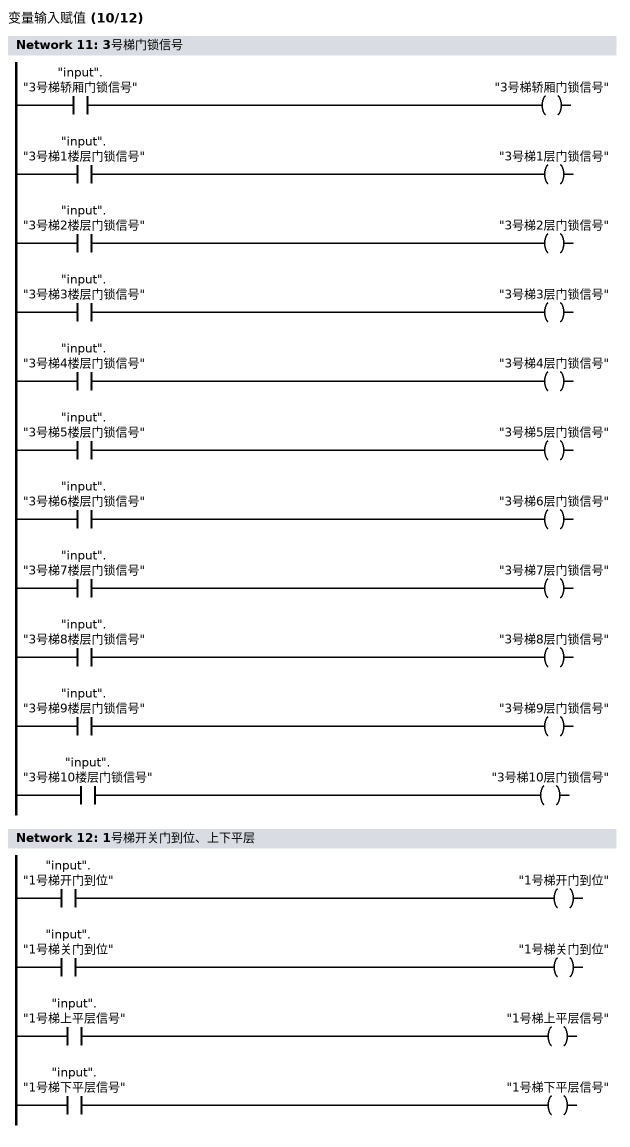
   RUNG wire#powerrail
      Contact( "input"."3号梯轿厢门锁信号" )
      Coil( "3号梯轿厢门锁信号" )
   END_RUNG
   RUNG wire#powerrail
      Contact( "input"."3号梯1楼层门锁信号" )
      Coil( "3号梯1层门锁信号" )
   END_RUNG
   RUNG wire#powerrail
      Contact( "input"."3号梯2楼层门锁信号" )
      Coil( "3号梯2层门锁信号" )
   END_RUNG
   RUNG wire#powerrail
      Contact( "input"."3号梯3楼层门锁信号" )
      Coil( "3号梯3层门锁信号" )
   END_RUNG
   RUNG wire#powerrail
      Contact( "input"."3号梯4楼层门锁信号" )
      Coil( "3号梯4层门锁信号" )
   END_RUNG
   RUNG wire#powerrail
      Contact( "input"."3号梯5楼层门锁信号" )
      Coil( "3号梯5层门锁信号" )
   END_RUNG
   RUNG wire#powerrail
      Contact( "input"."3号梯6楼层门锁信号" )
      Coil( "3号梯6层门锁信号" )
   END_RUNG
   RUNG wire#powerrail
      Contact( "input"."3号梯7楼层门锁信号" )
      Coil( "3号梯7层门锁信号" )
   END_RUNG
   RUNG wire#powerrail
      Contact( "input"."3号梯8楼层门锁信号" )
      Coil( "3号梯8层门锁信号" )
   END_RUNG
   RUNG wire#powerrail
      Contact( "input"."3号梯9楼层门锁信号" )
      Coil( "3号梯9层门锁信号" )
   END_RUNG
   RUNG wire#powerrail
      Contact( "input"."3号梯10楼层门锁信号" )
      Coil( "3号梯10层门锁信号" )
   END_RUNG
   // the same network as SCL:
   "3号梯轿厢门锁信号" := "input"."3号梯轿厢门锁信号";
   "3号梯1层门锁信号" := "input"."3号梯1楼层门锁信号";
   "3号梯2层门锁信号" := "input"."3号梯2楼层门锁信号";
   "3号梯3层门锁信号" := "input"."3号梯3楼层门锁信号";
   "3号梯4层门锁信号" := "input"."3号梯4楼层门锁信号";
   "3号梯5层门锁信号" := "input"."3号梯5楼层门锁信号";
   "3号梯6层门锁信号" := "input"."3号梯6楼层门锁信号";
   "3号梯7层门锁信号" := "input"."3号梯7楼层门锁信号";
   "3号梯8层门锁信号" := "input"."3号梯8楼层门锁信号";
   "3号梯9层门锁信号" := "input"."3号梯9楼层门锁信号";
   "3号梯10层门锁信号" := "input"."3号梯10楼层门锁信号";
END_REGION

REGION Network 12: 1号梯开关门到位、上下平层
   RUNG wire#powerrail
      Contact( "input"."1号梯开门到位" )
      Coil( "1号梯开门到位" )
   END_RUNG
   RUNG wire#powerrail
      Contact( "input"."1号梯关门到位" )
      Coil( "1号梯关门到位" )
   END_RUNG
   RUNG wire#powerrail
      Contact( "input"."1号梯上平层信号" )
      Coil( "1号梯上平层信号" )
   END_RUNG
   RUNG wire#powerrail
      Contact( "input"."1号梯下平层信号" )
      Coil( "1号梯下平层信号" )
   END_RUNG
   // the same network as SCL:
   "1号梯开门到位" := "input"."1号梯开门到位";
   "1号梯关门到位" := "input"."1号梯关门到位";
   "1号梯上平层信号" := "input"."1号梯上平层信号";
   "1号梯下平层信号" := "input"."1号梯下平层信号";
END_REGION

REGION Network 13: 2号梯开关门到位、上下平层
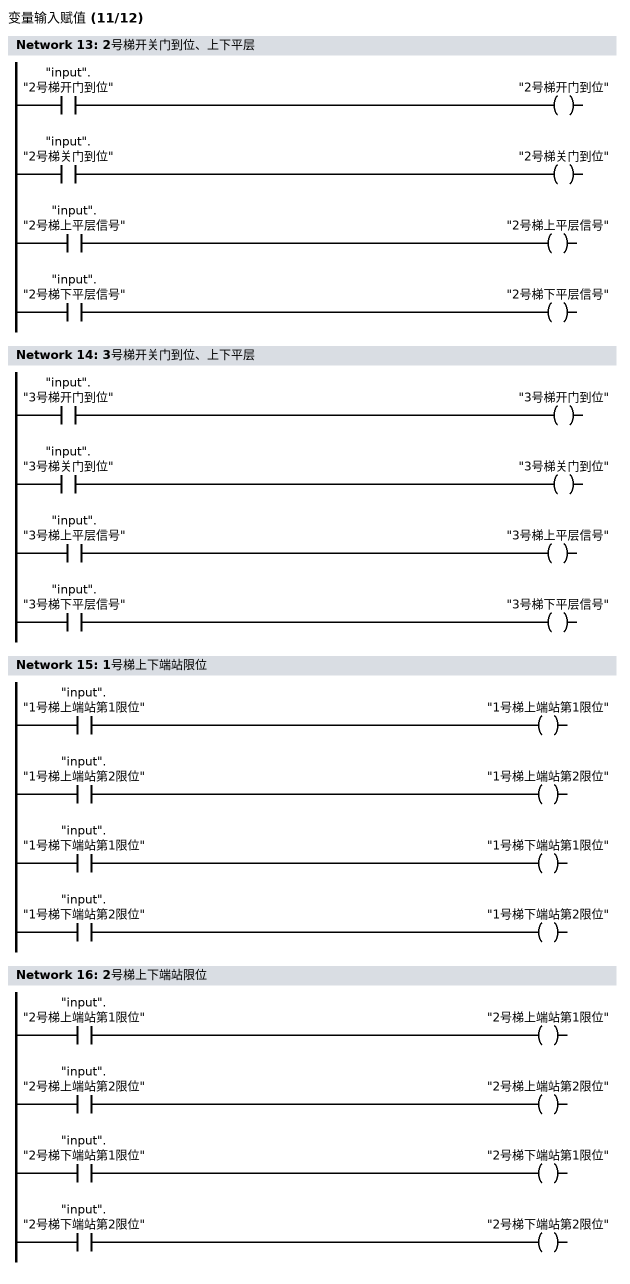
   RUNG wire#powerrail
      Contact( "input"."2号梯开门到位" )
      Coil( "2号梯开门到位" )
   END_RUNG
   RUNG wire#powerrail
      Contact( "input"."2号梯关门到位" )
      Coil( "2号梯关门到位" )
   END_RUNG
   RUNG wire#powerrail
      Contact( "input"."2号梯上平层信号" )
      Coil( "2号梯上平层信号" )
   END_RUNG
   RUNG wire#powerrail
      Contact( "input"."2号梯下平层信号" )
      Coil( "2号梯下平层信号" )
   END_RUNG
   // the same network as SCL:
   "2号梯开门到位" := "input"."2号梯开门到位";
   "2号梯关门到位" := "input"."2号梯关门到位";
   "2号梯上平层信号" := "input"."2号梯上平层信号";
   "2号梯下平层信号" := "input"."2号梯下平层信号";
END_REGION

REGION Network 14: 3号梯开关门到位、上下平层
   RUNG wire#powerrail
      Contact( "input"."3号梯开门到位" )
      Coil( "3号梯开门到位" )
   END_RUNG
   RUNG wire#powerrail
      Contact( "input"."3号梯关门到位" )
      Coil( "3号梯关门到位" )
   END_RUNG
   RUNG wire#powerrail
      Contact( "input"."3号梯上平层信号" )
      Coil( "3号梯上平层信号" )
   END_RUNG
   RUNG wire#powerrail
      Contact( "input"."3号梯下平层信号" )
      Coil( "3号梯下平层信号" )
   END_RUNG
   // the same network as SCL:
   "3号梯开门到位" := "input"."3号梯开门到位";
   "3号梯关门到位" := "input"."3号梯关门到位";
   "3号梯上平层信号" := "input"."3号梯上平层信号";
   "3号梯下平层信号" := "input"."3号梯下平层信号";
END_REGION

REGION Network 15: 1号梯上下端站限位
   RUNG wire#powerrail
      Contact( "input"."1号梯上端站第1限位" )
      Coil( "1号梯上端站第1限位" )
   END_RUNG
   RUNG wire#powerrail
      Contact( "input"."1号梯上端站第2限位" )
      Coil( "1号梯上端站第2限位" )
   END_RUNG
   RUNG wire#powerrail
      Contact( "input"."1号梯下端站第1限位" )
      Coil( "1号梯下端站第1限位" )
   END_RUNG
   RUNG wire#powerrail
      Contact( "input"."1号梯下端站第2限位" )
      Coil( "1号梯下端站第2限位" )
   END_RUNG
   // the same network as SCL:
   "1号梯上端站第1限位" := "input"."1号梯上端站第1限位";
   "1号梯上端站第2限位" := "input"."1号梯上端站第2限位";
   "1号梯下端站第1限位" := "input"."1号梯下端站第1限位";
   "1号梯下端站第2限位" := "input"."1号梯下端站第2限位";
END_REGION

REGION Network 16: 2号梯上下端站限位
   RUNG wire#powerrail
      Contact( "input"."2号梯上端站第1限位" )
      Coil( "2号梯上端站第1限位" )
   END_RUNG
   RUNG wire#powerrail
      Contact( "input"."2号梯上端站第2限位" )
      Coil( "2号梯上端站第2限位" )
   END_RUNG
   RUNG wire#powerrail
      Contact( "input"."2号梯下端站第1限位" )
      Coil( "2号梯下端站第1限位" )
   END_RUNG
   RUNG wire#powerrail
      Contact( "input"."2号梯下端站第2限位" )
      Coil( "2号梯下端站第2限位" )
   END_RUNG
   // the same network as SCL:
   "2号梯上端站第1限位" := "input"."2号梯上端站第1限位";
   "2号梯上端站第2限位" := "input"."2号梯上端站第2限位";
   "2号梯下端站第1限位" := "input"."2号梯下端站第1限位";
   "2号梯下端站第2限位" := "input"."2号梯下端站第2限位";
END_REGION

REGION Network 17: 3号梯上下端站限位
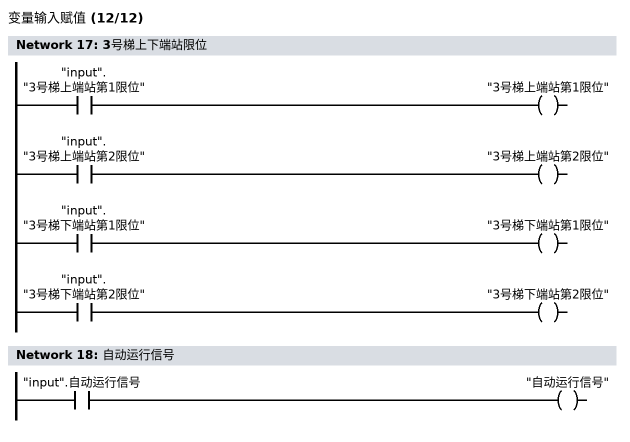
   RUNG wire#powerrail
      Contact( "input"."3号梯上端站第1限位" )
      Coil( "3号梯上端站第1限位" )
   END_RUNG
   RUNG wire#powerrail
      Contact( "input"."3号梯上端站第2限位" )
      Coil( "3号梯上端站第2限位" )
   END_RUNG
   RUNG wire#powerrail
      Contact( "input"."3号梯下端站第1限位" )
      Coil( "3号梯下端站第1限位" )
   END_RUNG
   RUNG wire#powerrail
      Contact( "input"."3号梯下端站第2限位" )
      Coil( "3号梯下端站第2限位" )
   END_RUNG
   // the same network as SCL:
   "3号梯上端站第1限位" := "input"."3号梯上端站第1限位";
   "3号梯上端站第2限位" := "input"."3号梯上端站第2限位";
   "3号梯下端站第1限位" := "input"."3号梯下端站第1限位";
   "3号梯下端站第2限位" := "input"."3号梯下端站第2限位";
END_REGION

REGION Network 18: 自动运行信号
   RUNG wire#powerrail
      Contact( "input".自动运行信号 )
      Coil( "自动运行信号" )
   END_RUNG
   // the same network as SCL:
   "自动运行信号" := "input".自动运行信号;
END_REGION
END_FUNCTION

FUNCTION "FC_GC_Score" : Int   // FC4, SCL
{ S7_Optimized_Access := 'TRUE' }
   VAR_INPUT
      ReqFloor : Int;
      ReqDir : Int;
      LiftFloor : Int;
      LiftDir : Int;
      LiftRunning : Bool;
      LiftLoadPercent : Int;
      TaskCount : Int;
      AheadTaskCount : Int;
      CanUse : Bool;
      W_Distance : Int;
      W_Direction : Int;
      W_Task : Int;
      W_AheadTask : Int;
      W_LoadPercent : Real;
      empty : Int;
   END_VAR
   VAR_TEMP
      tmpDist : Int;
      tmpScore : Int;
   END_VAR
BEGIN
   // ==================================================
   // FC_GC_Score 优化版
   //
   // 方向定义：
   //    1 = 上行
   //    0 = 停止/空闲
   //   -1 = 下行
   //
   // 评分越低，派梯优先级越高
   // ==================================================


   // ==================================================
   // 1. 可用性及输入有效性检查
   // ==================================================
   IF (NOT #CanUse)
       OR (#ReqFloor < 1)
       OR (#ReqFloor > 10)
       OR (#LiftFloor < 1)
       OR (#LiftFloor > 10)
       OR ((#ReqDir <> 1) AND (#ReqDir <> -1))
       OR (
       (#LiftDir <> -1)
       AND (#LiftDir <> 0)
       AND (#LiftDir <> 1)
       ) THEN

       // 32000表示该电梯不可参与派梯
       #FC_GC_Score := 32000;

   ELSE

       // ==================================================
       // 2. 距离评分
       // ==================================================
       #tmpDist := ABS(#ReqFloor - #LiftFloor);

       #tmpScore :=
       #tmpDist * #W_Distance;


       // ==================================================
       // 3. 方向和路线评分
       // ==================================================

       // --------------------------------------------------
       // 3.1 LiftDir = 0：停止或空闲
       // --------------------------------------------------
       IF #LiftDir = 0 THEN

           // 所有方向为0的电梯均获得空闲奖励
           // 不限制电梯所在楼层
           #tmpScore :=
           #tmpScore - #empty;


           // --------------------------------------------------
           // 3.2 电梯运行方向与外呼方向相同
           // --------------------------------------------------
       ELSIF #LiftDir = #ReqDir THEN

           // 上行梯：请求楼层在当前楼层上方或同层
           // 下行梯：请求楼层在当前楼层下方或同层
           IF
               (
               (#LiftDir = 1)
               AND (#ReqFloor >= #LiftFloor)
               )
               OR
               (
               (#LiftDir = -1)
               AND (#ReqFloor <= #LiftFloor)
               ) THEN

               // 同方向且请求在运行前方，属于顺路
               #tmpScore := #tmpScore + 0;

           ELSE

               // 方向相同，但是已经越过请求楼层
               // 必须完成当前路线后换向返回
               #tmpScore :=
               #tmpScore
               + (#W_Direction * 2);

               // 增加部分返回距离惩罚
               #tmpScore :=
               #tmpScore
               + (
               #tmpDist
               * #W_Distance
               / 2
               );

           END_IF;


           // --------------------------------------------------
           // 3.3 电梯运行方向与外呼方向相反
           // --------------------------------------------------
       ELSE

           // 判断请求楼层是否位于电梯当前运动前方
           IF
               (
               (#LiftDir = 1)
               AND (#ReqFloor >= #LiftFloor)
               )
               OR
               (
               (#LiftDir = -1)
               AND (#ReqFloor <= #LiftFloor)
               ) THEN

               // 请求楼层位于当前运行前方，
               // 但是乘客请求方向与电梯方向相反
               #tmpScore :=
               #tmpScore
               + (#W_Direction * 2);

           ELSE

               // 请求楼层位于当前运行后方，
               // 同时乘客请求方向也与电梯方向相反
               // 属于最不利的派梯情况
               #tmpScore :=
               #tmpScore
               + (#W_Direction * 3);

               // 增加部分绕行距离惩罚
               #tmpScore :=
               #tmpScore
               + (
               #tmpDist
               * #W_Distance
               / 2
               );

           END_IF;

       END_IF;


       // ==================================================
       // 4. 当前总任务数量惩罚
       // ==================================================
       IF #TaskCount > 0 THEN

           #tmpScore :=
           #tmpScore
           + (#TaskCount * #W_Task);

       END_IF;


       // ==================================================
       // 5. 当前运行前方任务数量惩罚
       // ==================================================
       IF #AheadTaskCount > 0 THEN

           #tmpScore :=
           #tmpScore
           + (
           #AheadTaskCount
           * #W_AheadTask
           );

       END_IF;


       // ==================================================
       // 6. 载重量基础评分
       // ==================================================
       IF #LiftLoadPercent > 0 THEN

           #tmpScore :=
           #tmpScore
           + REAL_TO_INT(
                         INT_TO_REAL(#LiftLoadPercent)
                         * #W_LoadPercent
           );

       END_IF;


       // ==================================================
       // 7. 高载重附加惩罚
       // ==================================================
       IF #LiftLoadPercent >= 90 THEN

           // 载重量达到90%以上
           #tmpScore :=
           #tmpScore + #W_Direction;

       ELSIF #LiftLoadPercent >= 75 THEN

           // 载重量达到75%以上
           #tmpScore :=
           #tmpScore + (#W_Direction / 2);

       END_IF;


       // ==================================================
       // 8. 同层空闲电梯额外奖励
       // ==================================================
       IF (#tmpDist = 0)
           AND (#LiftDir = 0) THEN

           // 已经获得普通空闲奖励，
           // 同层空闲时再增加一次奖励
           #tmpScore :=
           #tmpScore
           - (#W_Direction / 2);

       END_IF;


       // ==================================================
       // 9. 最终评分范围保护
       // ==================================================
       IF #tmpScore < 0 THEN

           #tmpScore := 0;

       ELSIF #tmpScore > 31999 THEN

           // 32000专门保留给不可用电梯
           #tmpScore := 31999;

       END_IF;


       // ==================================================
       // 10. 返回评分结果
       // ==================================================
       #FC_GC_Score := #tmpScore;

   END_IF;
END_FUNCTION

FUNCTION "FC_GC_IO_Map" : Void   // FC5, SCL
{ S7_Optimized_Access := 'TRUE' }
BEGIN
      // ==================================================
      // 1. 鏃犳晥妤煎眰淇濇姢
      // ==================================================
      "DB_GC".HallUpBtn[10] := FALSE;
      "DB_GC".HallDownBtn[1] := FALSE;


      // ==================================================
      // 2. 鏆傛椂娌℃湁杞藉鐜囧拰鍔熺巼锛屽氨鍏堢粰榛樿鍊?
       // ==================================================
      "DB_GC".LiftLoadPercent[1] := 0;
      "DB_GC".LiftLoadPercent[2] := 0;
      "DB_GC".LiftLoadPercent[3] := 0;

      "DB_GC".LiftPower_kW[1] := 0.0;
      "DB_GC".LiftPower_kW[2] := 0.0;
      "DB_GC".LiftPower_kW[3] := 0.0;


      // ==================================================
      // 3. 缇ゆ帶浣胯兘 / 閿佹 / 绂佺敤
      // 鍚庨潰鎺?WINCC 鏃跺啀鏀规垚 HMI 鍙橀噺
      // ==================================================
      "DB_GC".LiftGroupEnable[1] := TRUE;
      "DB_GC".LiftGroupEnable[2] := TRUE;
      "DB_GC".LiftGroupEnable[3] := TRUE;

      "DB_GC".LiftLocked[1] := FALSE;
      "DB_GC".LiftLocked[2] := FALSE;
      "DB_GC".LiftLocked[3] := FALSE;

      "DB_GC".LiftDisabled[1] := FALSE;
      "DB_GC".LiftDisabled[2] := FALSE;
      "DB_GC".LiftDisabled[3] := FALSE;


      // ==================================================
      // 4. 缇ゆ帶妯″紡
      // 0鏅€氾紝1涓婄彮楂樺嘲锛?涓嬬彮楂樺嘲锛?鍗堥楂樺嘲锛?涓夊垎鍖?
       // ==================================================
      "DB_GC".GroupMode := 0;


      // ==================================================
      // 5. 涔樻鏃堕棿缁熻锛屾殏鏃朵笉鐢?
       // ==================================================
      "DB_GC".RideFinishPulse[1] := FALSE;
      "DB_GC".RideFinishPulse[2] := FALSE;
      "DB_GC".RideFinishPulse[3] := FALSE;

      "DB_GC".RideTimeSample_s[1] := 0.0;
      "DB_GC".RideTimeSample_s[2] := 0.0;
      "DB_GC".RideTimeSample_s[3] := 0.0;
END_FUNCTION

FUNCTION "消防模式" : Void   // FC6, LAD
{ S7_Optimized_Access := 'TRUE' }
VERSION : 0.1
   VAR_TEMP   // added for the SCL form of the ladder/FBD networks
      _w1 : Bool;
   END_VAR
BEGIN

REGION Network 1: 指示灯reset
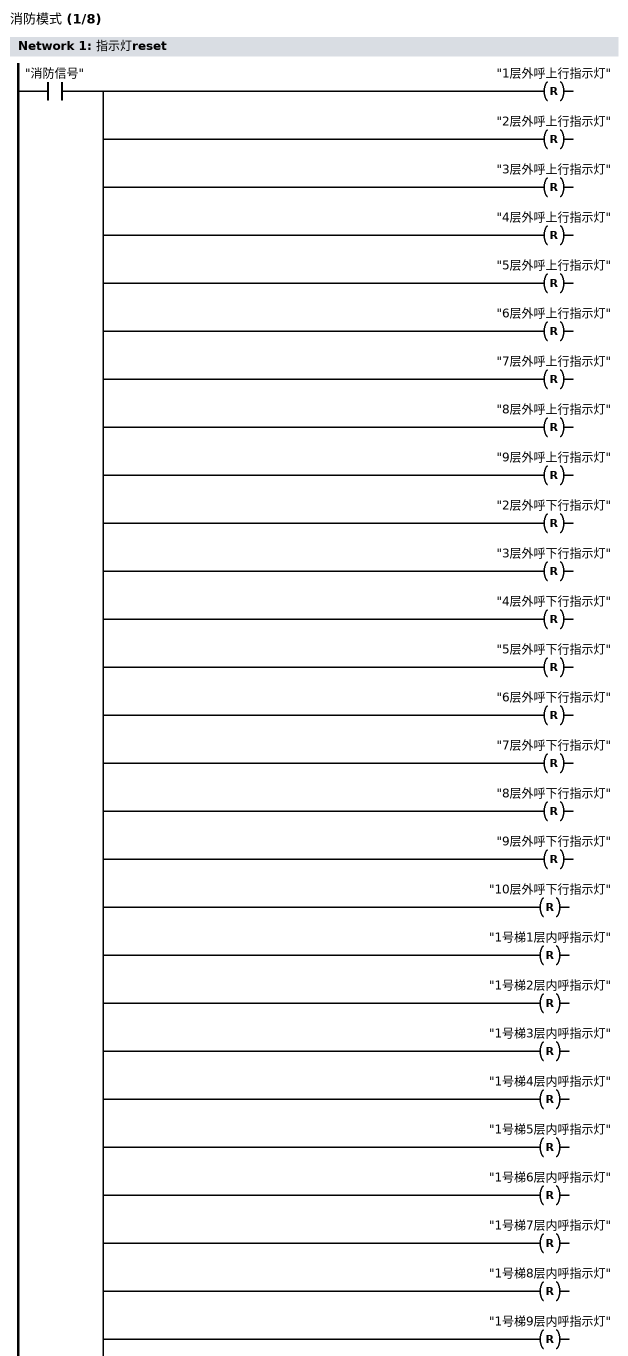
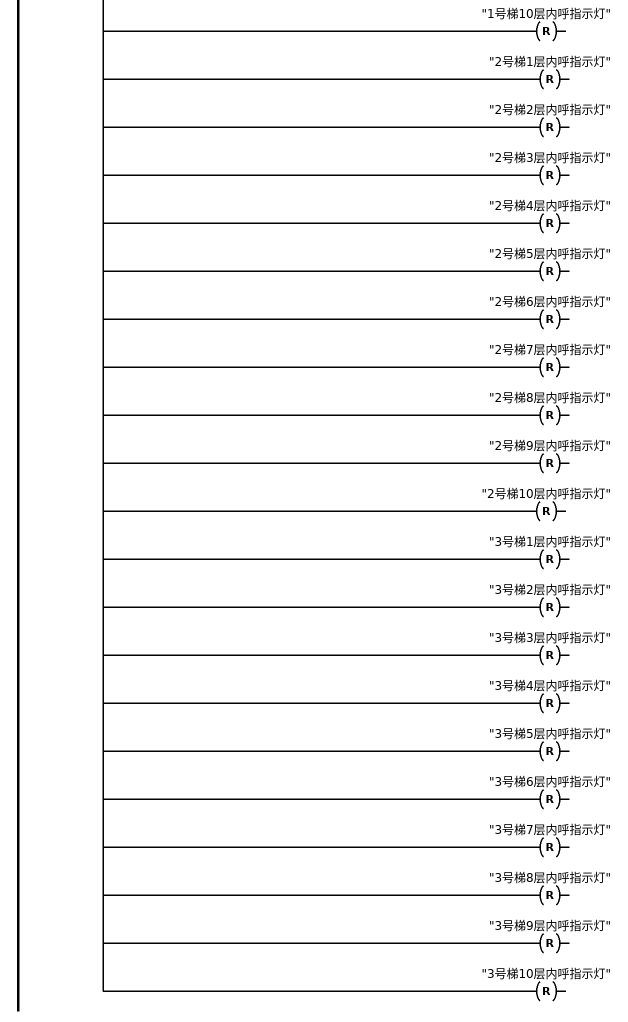
   RUNG wire#powerrail
      Contact( "消防信号" )
      wire#w1
      R_Coil( "1层外呼上行指示灯" )
   END_RUNG
   RUNG wire#w1
      R_Coil( "2层外呼上行指示灯" )
   END_RUNG
   RUNG wire#w1
      R_Coil( "3层外呼上行指示灯" )
   END_RUNG
   RUNG wire#w1
      R_Coil( "4层外呼上行指示灯" )
   END_RUNG
   RUNG wire#w1
      R_Coil( "5层外呼上行指示灯" )
   END_RUNG
   RUNG wire#w1
      R_Coil( "6层外呼上行指示灯" )
   END_RUNG
   RUNG wire#w1
      R_Coil( "7层外呼上行指示灯" )
   END_RUNG
   RUNG wire#w1
      R_Coil( "8层外呼上行指示灯" )
   END_RUNG
   RUNG wire#w1
      R_Coil( "9层外呼上行指示灯" )
   END_RUNG
   RUNG wire#w1
      R_Coil( "2层外呼下行指示灯" )
   END_RUNG
   RUNG wire#w1
      R_Coil( "3层外呼下行指示灯" )
   END_RUNG
   RUNG wire#w1
      R_Coil( "4层外呼下行指示灯" )
   END_RUNG
   RUNG wire#w1
      R_Coil( "5层外呼下行指示灯" )
   END_RUNG
   RUNG wire#w1
      R_Coil( "6层外呼下行指示灯" )
   END_RUNG
   RUNG wire#w1
      R_Coil( "7层外呼下行指示灯" )
   END_RUNG
   RUNG wire#w1
      R_Coil( "8层外呼下行指示灯" )
   END_RUNG
   RUNG wire#w1
      R_Coil( "9层外呼下行指示灯" )
   END_RUNG
   RUNG wire#w1
      R_Coil( "10层外呼下行指示灯" )
   END_RUNG
   RUNG wire#w1
      R_Coil( "1号梯1层内呼指示灯" )
   END_RUNG
   RUNG wire#w1
      R_Coil( "1号梯2层内呼指示灯" )
   END_RUNG
   RUNG wire#w1
      R_Coil( "1号梯3层内呼指示灯" )
   END_RUNG
   RUNG wire#w1
      R_Coil( "1号梯4层内呼指示灯" )
   END_RUNG
   RUNG wire#w1
      R_Coil( "1号梯5层内呼指示灯" )
   END_RUNG
   RUNG wire#w1
      R_Coil( "1号梯6层内呼指示灯" )
   END_RUNG
   RUNG wire#w1
      R_Coil( "1号梯7层内呼指示灯" )
   END_RUNG
   RUNG wire#w1
      R_Coil( "1号梯8层内呼指示灯" )
   END_RUNG
   RUNG wire#w1
      R_Coil( "1号梯9层内呼指示灯" )
   END_RUNG
   RUNG wire#w1
      R_Coil( "1号梯10层内呼指示灯" )
   END_RUNG
   RUNG wire#w1
      R_Coil( "2号梯1层内呼指示灯" )
   END_RUNG
   RUNG wire#w1
      R_Coil( "2号梯2层内呼指示灯" )
   END_RUNG
   RUNG wire#w1
      R_Coil( "2号梯3层内呼指示灯" )
   END_RUNG
   RUNG wire#w1
      R_Coil( "2号梯4层内呼指示灯" )
   END_RUNG
   RUNG wire#w1
      R_Coil( "2号梯5层内呼指示灯" )
   END_RUNG
   RUNG wire#w1
      R_Coil( "2号梯6层内呼指示灯" )
   END_RUNG
   RUNG wire#w1
      R_Coil( "2号梯7层内呼指示灯" )
   END_RUNG
   RUNG wire#w1
      R_Coil( "2号梯8层内呼指示灯" )
   END_RUNG
   RUNG wire#w1
      R_Coil( "2号梯9层内呼指示灯" )
   END_RUNG
   RUNG wire#w1
      R_Coil( "2号梯10层内呼指示灯" )
   END_RUNG
   RUNG wire#w1
      R_Coil( "3号梯1层内呼指示灯" )
   END_RUNG
   RUNG wire#w1
      R_Coil( "3号梯2层内呼指示灯" )
   END_RUNG
   RUNG wire#w1
      R_Coil( "3号梯3层内呼指示灯" )
   END_RUNG
   RUNG wire#w1
      R_Coil( "3号梯4层内呼指示灯" )
   END_RUNG
   RUNG wire#w1
      R_Coil( "3号梯5层内呼指示灯" )
   END_RUNG
   RUNG wire#w1
      R_Coil( "3号梯6层内呼指示灯" )
   END_RUNG
   RUNG wire#w1
      R_Coil( "3号梯7层内呼指示灯" )
   END_RUNG
   RUNG wire#w1
      R_Coil( "3号梯8层内呼指示灯" )
   END_RUNG
   RUNG wire#w1
      R_Coil( "3号梯9层内呼指示灯" )
   END_RUNG
   RUNG wire#w1
      R_Coil( "3号梯10层内呼指示灯" )
   END_RUNG
   // the same network as SCL:
   IF "消防信号" THEN
       "1层外呼上行指示灯" := FALSE;
       "2层外呼上行指示灯" := FALSE;
       "3层外呼上行指示灯" := FALSE;
       "4层外呼上行指示灯" := FALSE;
       "5层外呼上行指示灯" := FALSE;
       "6层外呼上行指示灯" := FALSE;
       "7层外呼上行指示灯" := FALSE;
       "8层外呼上行指示灯" := FALSE;
       "9层外呼上行指示灯" := FALSE;
       "2层外呼下行指示灯" := FALSE;
       "3层外呼下行指示灯" := FALSE;
       "4层外呼下行指示灯" := FALSE;
       "5层外呼下行指示灯" := FALSE;
       "6层外呼下行指示灯" := FALSE;
       "7层外呼下行指示灯" := FALSE;
       "8层外呼下行指示灯" := FALSE;
       "9层外呼下行指示灯" := FALSE;
       "10层外呼下行指示灯" := FALSE;
       "1号梯1层内呼指示灯" := FALSE;
       "1号梯2层内呼指示灯" := FALSE;
       "1号梯3层内呼指示灯" := FALSE;
       "1号梯4层内呼指示灯" := FALSE;
       "1号梯5层内呼指示灯" := FALSE;
       "1号梯6层内呼指示灯" := FALSE;
       "1号梯7层内呼指示灯" := FALSE;
       "1号梯8层内呼指示灯" := FALSE;
       "1号梯9层内呼指示灯" := FALSE;
       "1号梯10层内呼指示灯" := FALSE;
       "2号梯1层内呼指示灯" := FALSE;
       "2号梯2层内呼指示灯" := FALSE;
       "2号梯3层内呼指示灯" := FALSE;
       "2号梯4层内呼指示灯" := FALSE;
       "2号梯5层内呼指示灯" := FALSE;
       "2号梯6层内呼指示灯" := FALSE;
       "2号梯7层内呼指示灯" := FALSE;
       "2号梯8层内呼指示灯" := FALSE;
       "2号梯9层内呼指示灯" := FALSE;
       "2号梯10层内呼指示灯" := FALSE;
       "3号梯1层内呼指示灯" := FALSE;
       "3号梯2层内呼指示灯" := FALSE;
       "3号梯3层内呼指示灯" := FALSE;
       "3号梯4层内呼指示灯" := FALSE;
       "3号梯5层内呼指示灯" := FALSE;
       "3号梯6层内呼指示灯" := FALSE;
       "3号梯7层内呼指示灯" := FALSE;
       "3号梯8层内呼指示灯" := FALSE;
       "3号梯9层内呼指示灯" := FALSE;
       "3号梯10层内呼指示灯" := FALSE;
   END_IF;
END_REGION

REGION Network 2: 群控输出reset
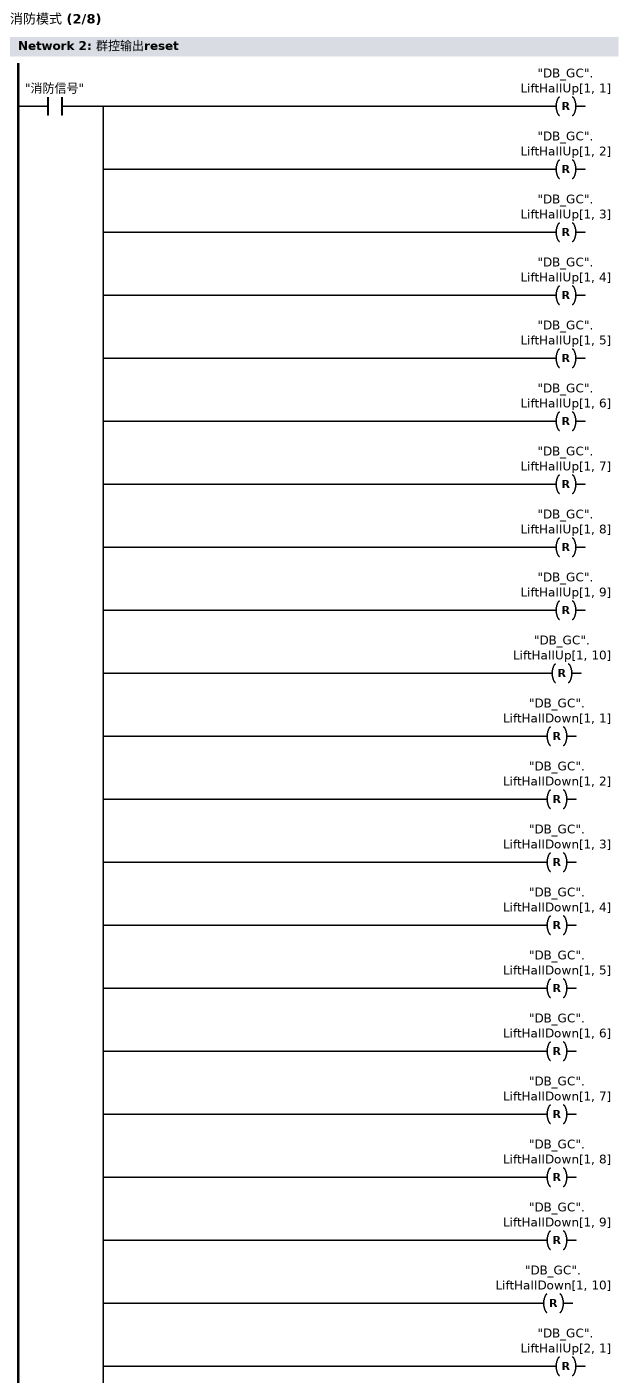
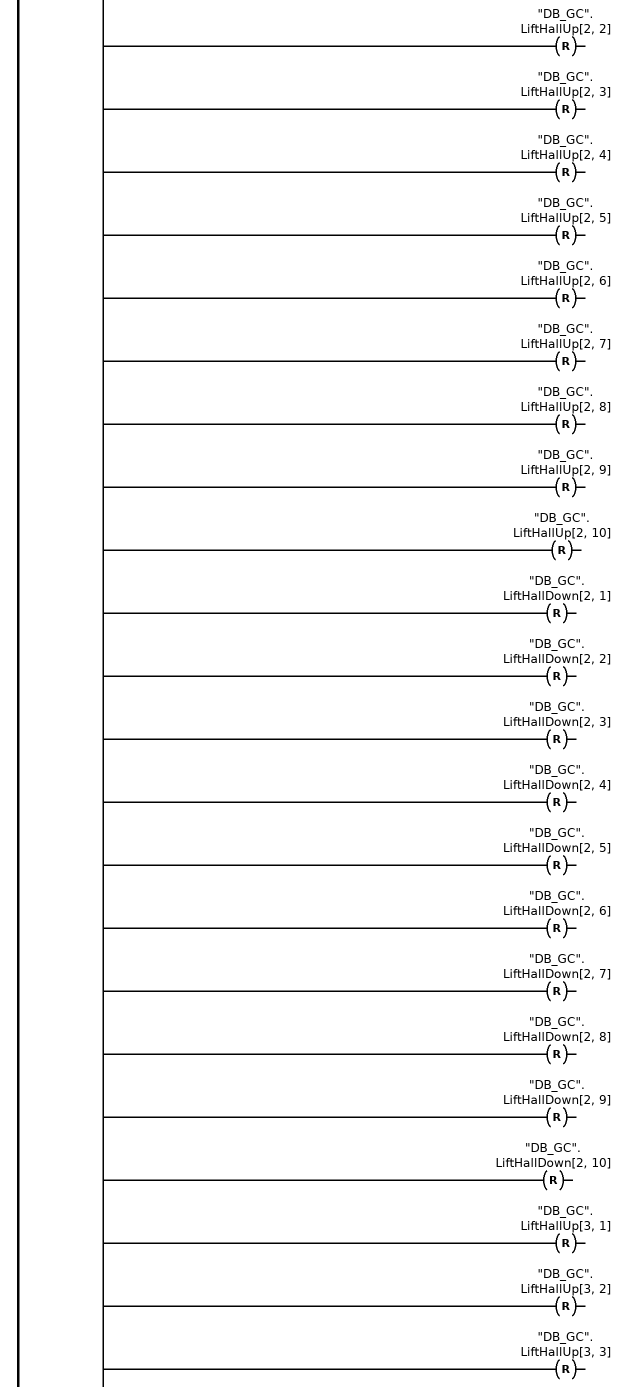
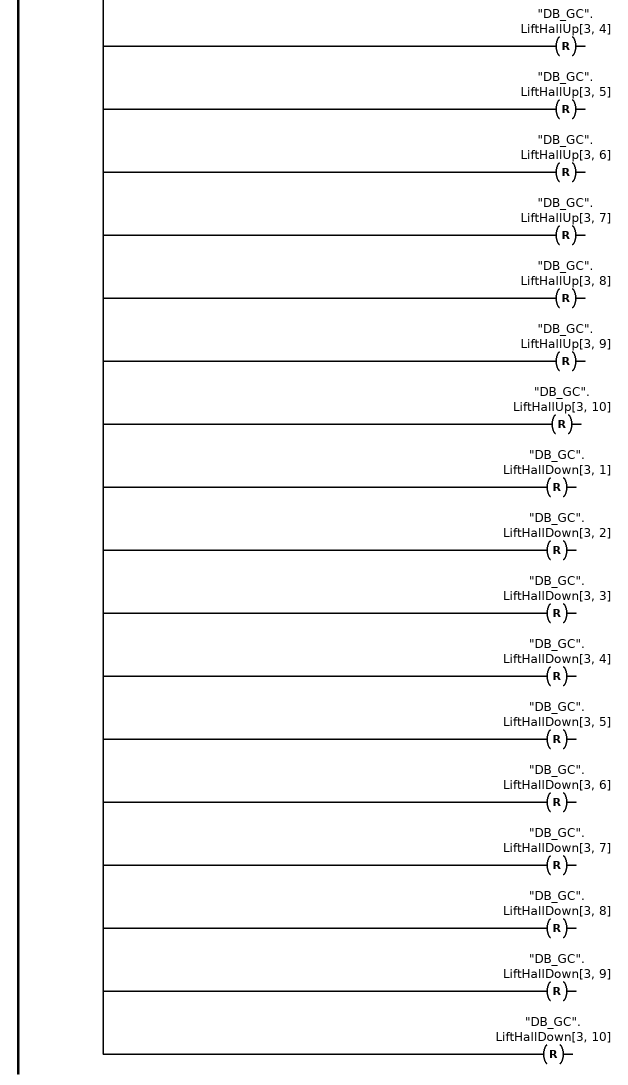
   RUNG wire#powerrail
      Contact( "消防信号" )
      wire#w1
      R_Coil( "DB_GC".LiftHallUp[1, 1] )
   END_RUNG
   RUNG wire#w1
      R_Coil( "DB_GC".LiftHallUp[1, 2] )
   END_RUNG
   RUNG wire#w1
      R_Coil( "DB_GC".LiftHallUp[1, 3] )
   END_RUNG
   RUNG wire#w1
      R_Coil( "DB_GC".LiftHallUp[1, 4] )
   END_RUNG
   RUNG wire#w1
      R_Coil( "DB_GC".LiftHallUp[1, 5] )
   END_RUNG
   RUNG wire#w1
      R_Coil( "DB_GC".LiftHallUp[1, 6] )
   END_RUNG
   RUNG wire#w1
      R_Coil( "DB_GC".LiftHallUp[1, 7] )
   END_RUNG
   RUNG wire#w1
      R_Coil( "DB_GC".LiftHallUp[1, 8] )
   END_RUNG
   RUNG wire#w1
      R_Coil( "DB_GC".LiftHallUp[1, 9] )
   END_RUNG
   RUNG wire#w1
      R_Coil( "DB_GC".LiftHallUp[1, 10] )
   END_RUNG
   RUNG wire#w1
      R_Coil( "DB_GC".LiftHallDown[1, 1] )
   END_RUNG
   RUNG wire#w1
      R_Coil( "DB_GC".LiftHallDown[1, 2] )
   END_RUNG
   RUNG wire#w1
      R_Coil( "DB_GC".LiftHallDown[1, 3] )
   END_RUNG
   RUNG wire#w1
      R_Coil( "DB_GC".LiftHallDown[1, 4] )
   END_RUNG
   RUNG wire#w1
      R_Coil( "DB_GC".LiftHallDown[1, 5] )
   END_RUNG
   RUNG wire#w1
      R_Coil( "DB_GC".LiftHallDown[1, 6] )
   END_RUNG
   RUNG wire#w1
      R_Coil( "DB_GC".LiftHallDown[1, 7] )
   END_RUNG
   RUNG wire#w1
      R_Coil( "DB_GC".LiftHallDown[1, 8] )
   END_RUNG
   RUNG wire#w1
      R_Coil( "DB_GC".LiftHallDown[1, 9] )
   END_RUNG
   RUNG wire#w1
      R_Coil( "DB_GC".LiftHallDown[1, 10] )
   END_RUNG
   RUNG wire#w1
      R_Coil( "DB_GC".LiftHallUp[2, 1] )
   END_RUNG
   RUNG wire#w1
      R_Coil( "DB_GC".LiftHallUp[2, 2] )
   END_RUNG
   RUNG wire#w1
      R_Coil( "DB_GC".LiftHallUp[2, 3] )
   END_RUNG
   RUNG wire#w1
      R_Coil( "DB_GC".LiftHallUp[2, 4] )
   END_RUNG
   RUNG wire#w1
      R_Coil( "DB_GC".LiftHallUp[2, 5] )
   END_RUNG
   RUNG wire#w1
      R_Coil( "DB_GC".LiftHallUp[2, 6] )
   END_RUNG
   RUNG wire#w1
      R_Coil( "DB_GC".LiftHallUp[2, 7] )
   END_RUNG
   RUNG wire#w1
      R_Coil( "DB_GC".LiftHallUp[2, 8] )
   END_RUNG
   RUNG wire#w1
      R_Coil( "DB_GC".LiftHallUp[2, 9] )
   END_RUNG
   RUNG wire#w1
      R_Coil( "DB_GC".LiftHallUp[2, 10] )
   END_RUNG
   RUNG wire#w1
      R_Coil( "DB_GC".LiftHallDown[2, 1] )
   END_RUNG
   RUNG wire#w1
      R_Coil( "DB_GC".LiftHallDown[2, 2] )
   END_RUNG
   RUNG wire#w1
      R_Coil( "DB_GC".LiftHallDown[2, 3] )
   END_RUNG
   RUNG wire#w1
      R_Coil( "DB_GC".LiftHallDown[2, 4] )
   END_RUNG
   RUNG wire#w1
      R_Coil( "DB_GC".LiftHallDown[2, 5] )
   END_RUNG
   RUNG wire#w1
      R_Coil( "DB_GC".LiftHallDown[2, 6] )
   END_RUNG
   RUNG wire#w1
      R_Coil( "DB_GC".LiftHallDown[2, 7] )
   END_RUNG
   RUNG wire#w1
      R_Coil( "DB_GC".LiftHallDown[2, 8] )
   END_RUNG
   RUNG wire#w1
      R_Coil( "DB_GC".LiftHallDown[2, 9] )
   END_RUNG
   RUNG wire#w1
      R_Coil( "DB_GC".LiftHallDown[2, 10] )
   END_RUNG
   RUNG wire#w1
      R_Coil( "DB_GC".LiftHallUp[3, 1] )
   END_RUNG
   RUNG wire#w1
      R_Coil( "DB_GC".LiftHallUp[3, 2] )
   END_RUNG
   RUNG wire#w1
      R_Coil( "DB_GC".LiftHallUp[3, 3] )
   END_RUNG
   RUNG wire#w1
      R_Coil( "DB_GC".LiftHallUp[3, 4] )
   END_RUNG
   RUNG wire#w1
      R_Coil( "DB_GC".LiftHallUp[3, 5] )
   END_RUNG
   RUNG wire#w1
      R_Coil( "DB_GC".LiftHallUp[3, 6] )
   END_RUNG
   RUNG wire#w1
      R_Coil( "DB_GC".LiftHallUp[3, 7] )
   END_RUNG
   RUNG wire#w1
      R_Coil( "DB_GC".LiftHallUp[3, 8] )
   END_RUNG
   RUNG wire#w1
      R_Coil( "DB_GC".LiftHallUp[3, 9] )
   END_RUNG
   RUNG wire#w1
      R_Coil( "DB_GC".LiftHallUp[3, 10] )
   END_RUNG
   RUNG wire#w1
      R_Coil( "DB_GC".LiftHallDown[3, 1] )
   END_RUNG
   RUNG wire#w1
      R_Coil( "DB_GC".LiftHallDown[3, 2] )
   END_RUNG
   RUNG wire#w1
      R_Coil( "DB_GC".LiftHallDown[3, 3] )
   END_RUNG
   RUNG wire#w1
      R_Coil( "DB_GC".LiftHallDown[3, 4] )
   END_RUNG
   RUNG wire#w1
      R_Coil( "DB_GC".LiftHallDown[3, 5] )
   END_RUNG
   RUNG wire#w1
      R_Coil( "DB_GC".LiftHallDown[3, 6] )
   END_RUNG
   RUNG wire#w1
      R_Coil( "DB_GC".LiftHallDown[3, 7] )
   END_RUNG
   RUNG wire#w1
      R_Coil( "DB_GC".LiftHallDown[3, 8] )
   END_RUNG
   RUNG wire#w1
      R_Coil( "DB_GC".LiftHallDown[3, 9] )
   END_RUNG
   RUNG wire#w1
      R_Coil( "DB_GC".LiftHallDown[3, 10] )
   END_RUNG
   // the same network as SCL:
   IF "消防信号" THEN
       "DB_GC".LiftHallUp[1, 1] := FALSE;
       "DB_GC".LiftHallUp[1, 2] := FALSE;
       "DB_GC".LiftHallUp[1, 3] := FALSE;
       "DB_GC".LiftHallUp[1, 4] := FALSE;
       "DB_GC".LiftHallUp[1, 5] := FALSE;
       "DB_GC".LiftHallUp[1, 6] := FALSE;
       "DB_GC".LiftHallUp[1, 7] := FALSE;
       "DB_GC".LiftHallUp[1, 8] := FALSE;
       "DB_GC".LiftHallUp[1, 9] := FALSE;
       "DB_GC".LiftHallUp[1, 10] := FALSE;
       "DB_GC".LiftHallDown[1, 1] := FALSE;
       "DB_GC".LiftHallDown[1, 2] := FALSE;
       "DB_GC".LiftHallDown[1, 3] := FALSE;
       "DB_GC".LiftHallDown[1, 4] := FALSE;
       "DB_GC".LiftHallDown[1, 5] := FALSE;
       "DB_GC".LiftHallDown[1, 6] := FALSE;
       "DB_GC".LiftHallDown[1, 7] := FALSE;
       "DB_GC".LiftHallDown[1, 8] := FALSE;
       "DB_GC".LiftHallDown[1, 9] := FALSE;
       "DB_GC".LiftHallDown[1, 10] := FALSE;
       "DB_GC".LiftHallUp[2, 1] := FALSE;
       "DB_GC".LiftHallUp[2, 2] := FALSE;
       "DB_GC".LiftHallUp[2, 3] := FALSE;
       "DB_GC".LiftHallUp[2, 4] := FALSE;
       "DB_GC".LiftHallUp[2, 5] := FALSE;
       "DB_GC".LiftHallUp[2, 6] := FALSE;
       "DB_GC".LiftHallUp[2, 7] := FALSE;
       "DB_GC".LiftHallUp[2, 8] := FALSE;
       "DB_GC".LiftHallUp[2, 9] := FALSE;
       "DB_GC".LiftHallUp[2, 10] := FALSE;
       "DB_GC".LiftHallDown[2, 1] := FALSE;
       "DB_GC".LiftHallDown[2, 2] := FALSE;
       "DB_GC".LiftHallDown[2, 3] := FALSE;
       "DB_GC".LiftHallDown[2, 4] := FALSE;
       "DB_GC".LiftHallDown[2, 5] := FALSE;
       "DB_GC".LiftHallDown[2, 6] := FALSE;
       "DB_GC".LiftHallDown[2, 7] := FALSE;
       "DB_GC".LiftHallDown[2, 8] := FALSE;
       "DB_GC".LiftHallDown[2, 9] := FALSE;
       "DB_GC".LiftHallDown[2, 10] := FALSE;
       "DB_GC".LiftHallUp[3, 1] := FALSE;
       "DB_GC".LiftHallUp[3, 2] := FALSE;
       "DB_GC".LiftHallUp[3, 3] := FALSE;
       "DB_GC".LiftHallUp[3, 4] := FALSE;
       "DB_GC".LiftHallUp[3, 5] := FALSE;
       "DB_GC".LiftHallUp[3, 6] := FALSE;
       "DB_GC".LiftHallUp[3, 7] := FALSE;
       "DB_GC".LiftHallUp[3, 8] := FALSE;
       "DB_GC".LiftHallUp[3, 9] := FALSE;
       "DB_GC".LiftHallUp[3, 10] := FALSE;
       "DB_GC".LiftHallDown[3, 1] := FALSE;
       "DB_GC".LiftHallDown[3, 2] := FALSE;
       "DB_GC".LiftHallDown[3, 3] := FALSE;
       "DB_GC".LiftHallDown[3, 4] := FALSE;
       "DB_GC".LiftHallDown[3, 5] := FALSE;
       "DB_GC".LiftHallDown[3, 6] := FALSE;
       "DB_GC".LiftHallDown[3, 7] := FALSE;
       "DB_GC".LiftHallDown[3, 8] := FALSE;
       "DB_GC".LiftHallDown[3, 9] := FALSE;
       "DB_GC".LiftHallDown[3, 10] := FALSE;
   END_IF;
END_REGION

REGION Network 3: 群控输入的reset
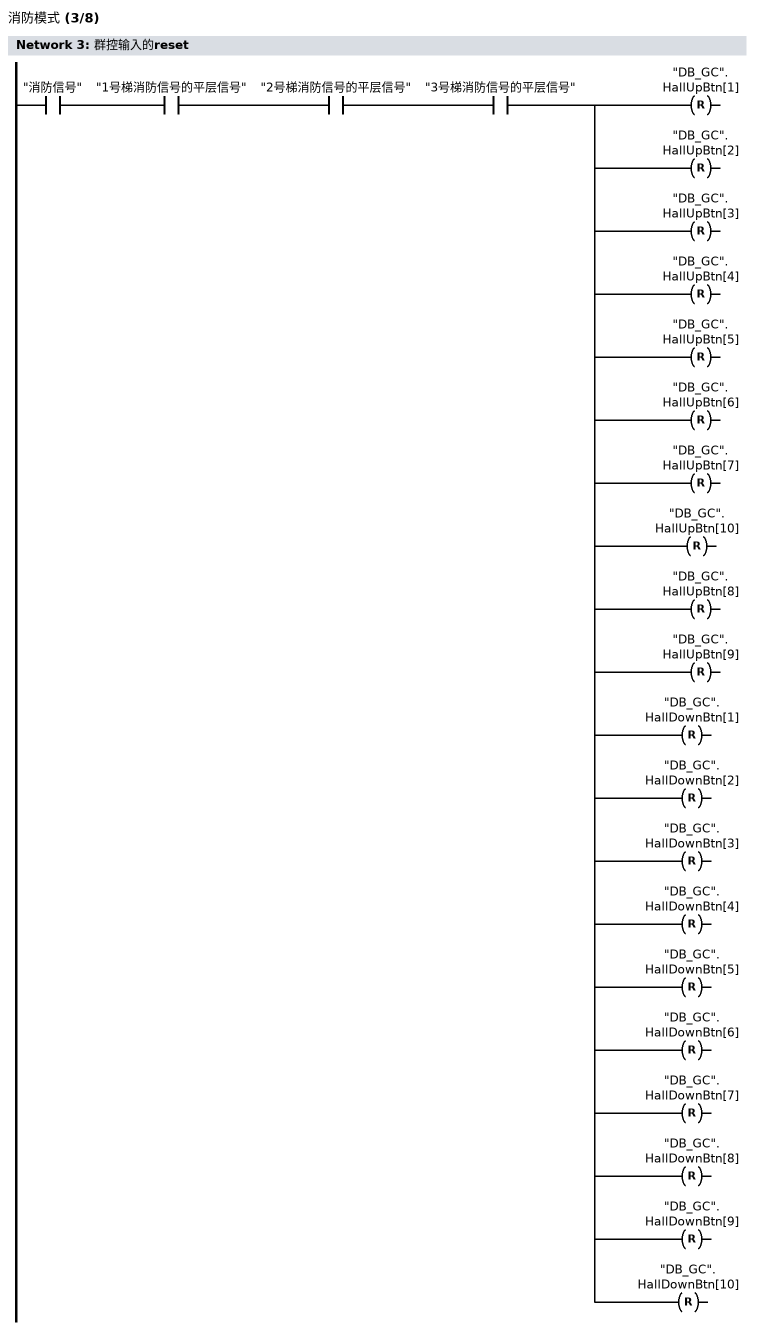
   RUNG wire#powerrail
      Contact( "消防信号" )
      Contact( "1号梯消防信号的平层信号" )
      Contact( "2号梯消防信号的平层信号" )
      Contact( "3号梯消防信号的平层信号" )
      wire#w1
      R_Coil( "DB_GC".HallUpBtn[1] )
   END_RUNG
   RUNG wire#w1
      R_Coil( "DB_GC".HallUpBtn[2] )
   END_RUNG
   RUNG wire#w1
      R_Coil( "DB_GC".HallUpBtn[3] )
   END_RUNG
   RUNG wire#w1
      R_Coil( "DB_GC".HallUpBtn[4] )
   END_RUNG
   RUNG wire#w1
      R_Coil( "DB_GC".HallUpBtn[5] )
   END_RUNG
   RUNG wire#w1
      R_Coil( "DB_GC".HallUpBtn[6] )
   END_RUNG
   RUNG wire#w1
      R_Coil( "DB_GC".HallUpBtn[7] )
   END_RUNG
   RUNG wire#w1
      R_Coil( "DB_GC".HallUpBtn[10] )
   END_RUNG
   RUNG wire#w1
      R_Coil( "DB_GC".HallUpBtn[8] )
   END_RUNG
   RUNG wire#w1
      R_Coil( "DB_GC".HallUpBtn[9] )
   END_RUNG
   RUNG wire#w1
      R_Coil( "DB_GC".HallDownBtn[1] )
   END_RUNG
   RUNG wire#w1
      R_Coil( "DB_GC".HallDownBtn[2] )
   END_RUNG
   RUNG wire#w1
      R_Coil( "DB_GC".HallDownBtn[3] )
   END_RUNG
   RUNG wire#w1
      R_Coil( "DB_GC".HallDownBtn[4] )
   END_RUNG
   RUNG wire#w1
      R_Coil( "DB_GC".HallDownBtn[5] )
   END_RUNG
   RUNG wire#w1
      R_Coil( "DB_GC".HallDownBtn[6] )
   END_RUNG
   RUNG wire#w1
      R_Coil( "DB_GC".HallDownBtn[7] )
   END_RUNG
   RUNG wire#w1
      R_Coil( "DB_GC".HallDownBtn[8] )
   END_RUNG
   RUNG wire#w1
      R_Coil( "DB_GC".HallDownBtn[9] )
   END_RUNG
   RUNG wire#w1
      R_Coil( "DB_GC".HallDownBtn[10] )
   END_RUNG
   // the same network as SCL:
   IF "消防信号" AND "1号梯消防信号的平层信号" AND "2号梯消防信号的平层信号" AND "3号梯消防信号的平层信号" THEN
       "DB_GC".HallUpBtn[1] := FALSE;
       "DB_GC".HallUpBtn[2] := FALSE;
       "DB_GC".HallUpBtn[3] := FALSE;
       "DB_GC".HallUpBtn[4] := FALSE;
       "DB_GC".HallUpBtn[5] := FALSE;
       "DB_GC".HallUpBtn[6] := FALSE;
       "DB_GC".HallUpBtn[7] := FALSE;
       "DB_GC".HallUpBtn[10] := FALSE;
       "DB_GC".HallUpBtn[8] := FALSE;
       "DB_GC".HallUpBtn[9] := FALSE;
       "DB_GC".HallDownBtn[1] := FALSE;
       "DB_GC".HallDownBtn[2] := FALSE;
       "DB_GC".HallDownBtn[3] := FALSE;
       "DB_GC".HallDownBtn[4] := FALSE;
       "DB_GC".HallDownBtn[5] := FALSE;
       "DB_GC".HallDownBtn[6] := FALSE;
       "DB_GC".HallDownBtn[7] := FALSE;
       "DB_GC".HallDownBtn[8] := FALSE;
       "DB_GC".HallDownBtn[9] := FALSE;
       "DB_GC".HallDownBtn[10] := FALSE;
   END_IF;
END_REGION

REGION Network 4: 群控输入的reset的promax
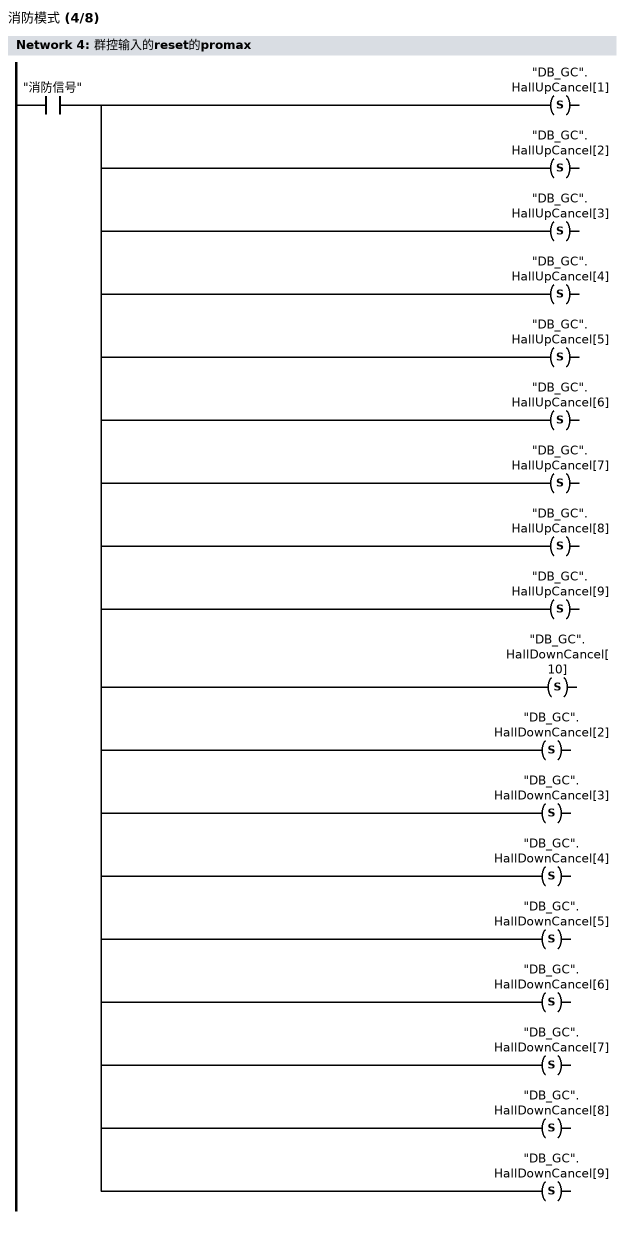
   RUNG wire#powerrail
      Contact( "消防信号" )
      wire#w1
      S_Coil( "DB_GC".HallUpCancel[1] )
   END_RUNG
   RUNG wire#w1
      S_Coil( "DB_GC".HallUpCancel[2] )
   END_RUNG
   RUNG wire#w1
      S_Coil( "DB_GC".HallUpCancel[3] )
   END_RUNG
   RUNG wire#w1
      S_Coil( "DB_GC".HallUpCancel[4] )
   END_RUNG
   RUNG wire#w1
      S_Coil( "DB_GC".HallUpCancel[5] )
   END_RUNG
   RUNG wire#w1
      S_Coil( "DB_GC".HallUpCancel[6] )
   END_RUNG
   RUNG wire#w1
      S_Coil( "DB_GC".HallUpCancel[7] )
   END_RUNG
   RUNG wire#w1
      S_Coil( "DB_GC".HallUpCancel[8] )
   END_RUNG
   RUNG wire#w1
      S_Coil( "DB_GC".HallUpCancel[9] )
   END_RUNG
   RUNG wire#w1
      S_Coil( "DB_GC".HallDownCancel[10] )
   END_RUNG
   RUNG wire#w1
      S_Coil( "DB_GC".HallDownCancel[2] )
   END_RUNG
   RUNG wire#w1
      S_Coil( "DB_GC".HallDownCancel[3] )
   END_RUNG
   RUNG wire#w1
      S_Coil( "DB_GC".HallDownCancel[4] )
   END_RUNG
   RUNG wire#w1
      S_Coil( "DB_GC".HallDownCancel[5] )
   END_RUNG
   RUNG wire#w1
      S_Coil( "DB_GC".HallDownCancel[6] )
   END_RUNG
   RUNG wire#w1
      S_Coil( "DB_GC".HallDownCancel[7] )
   END_RUNG
   RUNG wire#w1
      S_Coil( "DB_GC".HallDownCancel[8] )
   END_RUNG
   RUNG wire#w1
      S_Coil( "DB_GC".HallDownCancel[9] )
   END_RUNG
   // the same network as SCL:
   IF "消防信号" THEN
       "DB_GC".HallUpCancel[1] := TRUE;
       "DB_GC".HallUpCancel[2] := TRUE;
       "DB_GC".HallUpCancel[3] := TRUE;
       "DB_GC".HallUpCancel[4] := TRUE;
       "DB_GC".HallUpCancel[5] := TRUE;
       "DB_GC".HallUpCancel[6] := TRUE;
       "DB_GC".HallUpCancel[7] := TRUE;
       "DB_GC".HallUpCancel[8] := TRUE;
       "DB_GC".HallUpCancel[9] := TRUE;
       "DB_GC".HallDownCancel[10] := TRUE;
       "DB_GC".HallDownCancel[2] := TRUE;
       "DB_GC".HallDownCancel[3] := TRUE;
       "DB_GC".HallDownCancel[4] := TRUE;
       "DB_GC".HallDownCancel[5] := TRUE;
       "DB_GC".HallDownCancel[6] := TRUE;
       "DB_GC".HallDownCancel[7] := TRUE;
       "DB_GC".HallDownCancel[8] := TRUE;
       "DB_GC".HallDownCancel[9] := TRUE;
   END_IF;
END_REGION

REGION Network 5: 开门状态
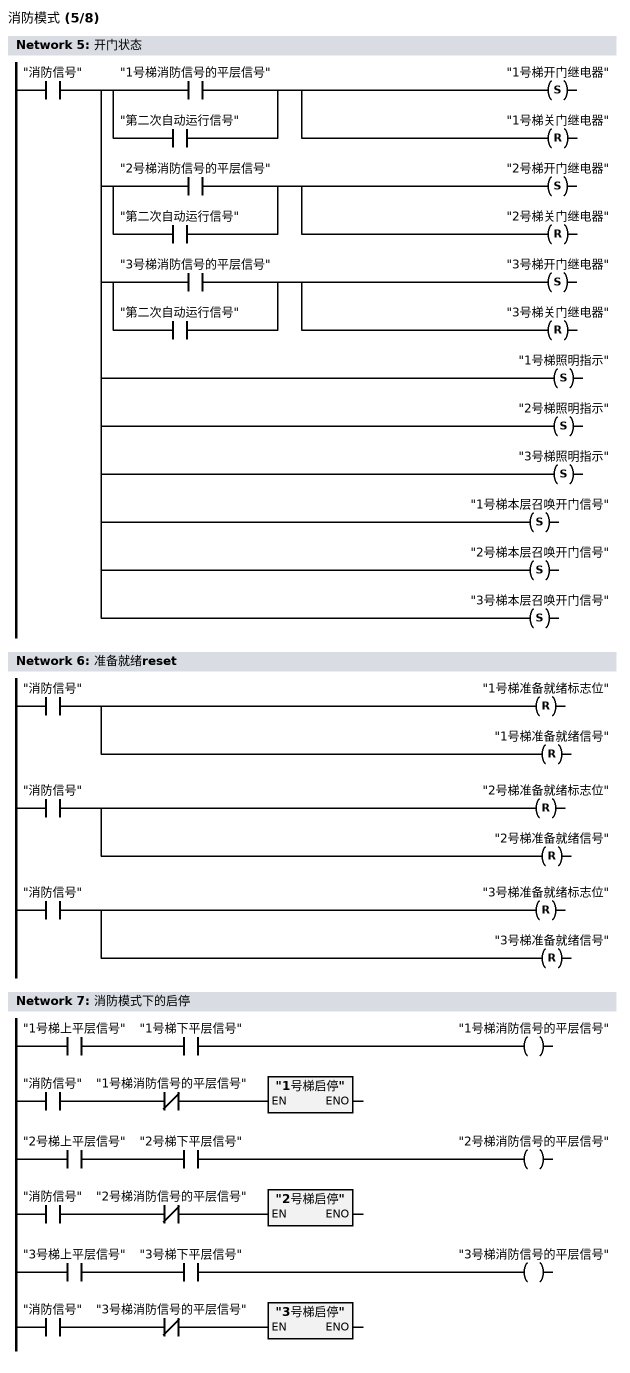
   RUNG wire#powerrail
      Contact( "消防信号" )
      wire#w1
      Contact( "1号梯消防信号的平层信号" )
      wire#w2
      S_Coil( "1号梯开门继电器" )
   END_RUNG
   RUNG wire#w1
      Contact( "第二次自动运行信号" )
   END_RUNG wire#w2
   RUNG wire#w2
      R_Coil( "1号梯关门继电器" )
   END_RUNG
   RUNG wire#w1
      Contact( "2号梯消防信号的平层信号" )
      wire#w3
      S_Coil( "2号梯开门继电器" )
   END_RUNG
   RUNG wire#w1
      Contact( "第二次自动运行信号" )
   END_RUNG wire#w3
   RUNG wire#w3
      R_Coil( "2号梯关门继电器" )
   END_RUNG
   RUNG wire#w1
      Contact( "3号梯消防信号的平层信号" )
      wire#w4
      S_Coil( "3号梯开门继电器" )
   END_RUNG
   RUNG wire#w1
      Contact( "第二次自动运行信号" )
   END_RUNG wire#w4
   RUNG wire#w4
      R_Coil( "3号梯关门继电器" )
   END_RUNG
   RUNG wire#w1
      S_Coil( "1号梯照明指示" )
   END_RUNG
   RUNG wire#w1
      S_Coil( "2号梯照明指示" )
   END_RUNG
   RUNG wire#w1
      S_Coil( "3号梯照明指示" )
   END_RUNG
   RUNG wire#w1
      S_Coil( "1号梯本层召唤开门信号" )
   END_RUNG
   RUNG wire#w1
      S_Coil( "2号梯本层召唤开门信号" )
   END_RUNG
   RUNG wire#w1
      S_Coil( "3号梯本层召唤开门信号" )
   END_RUNG
   // the same network as SCL:
   IF "消防信号" AND ("1号梯消防信号的平层信号" OR "第二次自动运行信号") THEN
       "1号梯开门继电器" := TRUE;
       "1号梯关门继电器" := FALSE;
   END_IF;
   IF "消防信号" AND ("2号梯消防信号的平层信号" OR "第二次自动运行信号") THEN
       "2号梯开门继电器" := TRUE;
       "2号梯关门继电器" := FALSE;
   END_IF;
   IF "消防信号" AND ("3号梯消防信号的平层信号" OR "第二次自动运行信号") THEN
       "3号梯开门继电器" := TRUE;
       "3号梯关门继电器" := FALSE;
   END_IF;
   IF "消防信号" THEN
       "1号梯照明指示" := TRUE;
       "2号梯照明指示" := TRUE;
       "3号梯照明指示" := TRUE;
       "1号梯本层召唤开门信号" := TRUE;
       "2号梯本层召唤开门信号" := TRUE;
       "3号梯本层召唤开门信号" := TRUE;
   END_IF;
END_REGION

REGION Network 6: 准备就绪reset
   RUNG wire#powerrail
      Contact( "消防信号" )
      wire#w1
      R_Coil( "1号梯准备就绪标志位" )
   END_RUNG
   RUNG wire#w1
      R_Coil( "1号梯准备就绪信号" )
   END_RUNG
   RUNG wire#powerrail
      Contact( "消防信号" )
      wire#w2
      R_Coil( "2号梯准备就绪标志位" )
   END_RUNG
   RUNG wire#w2
      R_Coil( "2号梯准备就绪信号" )
   END_RUNG
   RUNG wire#powerrail
      Contact( "消防信号" )
      wire#w3
      R_Coil( "3号梯准备就绪标志位" )
   END_RUNG
   RUNG wire#w3
      R_Coil( "3号梯准备就绪信号" )
   END_RUNG
   // the same network as SCL:
   IF "消防信号" THEN
       "1号梯准备就绪标志位" := FALSE;
       "1号梯准备就绪信号" := FALSE;
       "2号梯准备就绪标志位" := FALSE;
       "2号梯准备就绪信号" := FALSE;
       "3号梯准备就绪标志位" := FALSE;
       "3号梯准备就绪信号" := FALSE;
   END_IF;
END_REGION

REGION Network 7: 消防模式下的启停
   RUNG wire#powerrail
      Contact( "1号梯上平层信号" )
      Contact( "1号梯下平层信号" )
      Coil( "1号梯消防信号的平层信号" )
   END_RUNG
   RUNG wire#powerrail
      Contact( "消防信号" )
      I_Contact( "1号梯消防信号的平层信号" )
      "1号梯启停"()
   END_RUNG
   RUNG wire#powerrail
      Contact( "2号梯上平层信号" )
      Contact( "2号梯下平层信号" )
      Coil( "2号梯消防信号的平层信号" )
   END_RUNG
   RUNG wire#powerrail
      Contact( "消防信号" )
      I_Contact( "2号梯消防信号的平层信号" )
      "2号梯启停"()
   END_RUNG
   RUNG wire#powerrail
      Contact( "3号梯上平层信号" )
      Contact( "3号梯下平层信号" )
      Coil( "3号梯消防信号的平层信号" )
   END_RUNG
   RUNG wire#powerrail
      Contact( "消防信号" )
      I_Contact( "3号梯消防信号的平层信号" )
      "3号梯启停"()
   END_RUNG
   // the same network as SCL:
   "1号梯消防信号的平层信号" := "1号梯上平层信号" AND "1号梯下平层信号";
   IF "消防信号" AND NOT "1号梯消防信号的平层信号" THEN "1号梯启停"(); END_IF;
   "2号梯消防信号的平层信号" := "2号梯上平层信号" AND "2号梯下平层信号";
   IF "消防信号" AND NOT "2号梯消防信号的平层信号" THEN "2号梯启停"(); END_IF;
   "3号梯消防信号的平层信号" := "3号梯上平层信号" AND "3号梯下平层信号";
   IF "消防信号" AND NOT "3号梯消防信号的平层信号" THEN "3号梯启停"(); END_IF;
END_REGION

REGION Network 8: 给出初始化信号后，的上下行reset，关门，关门锁上下行
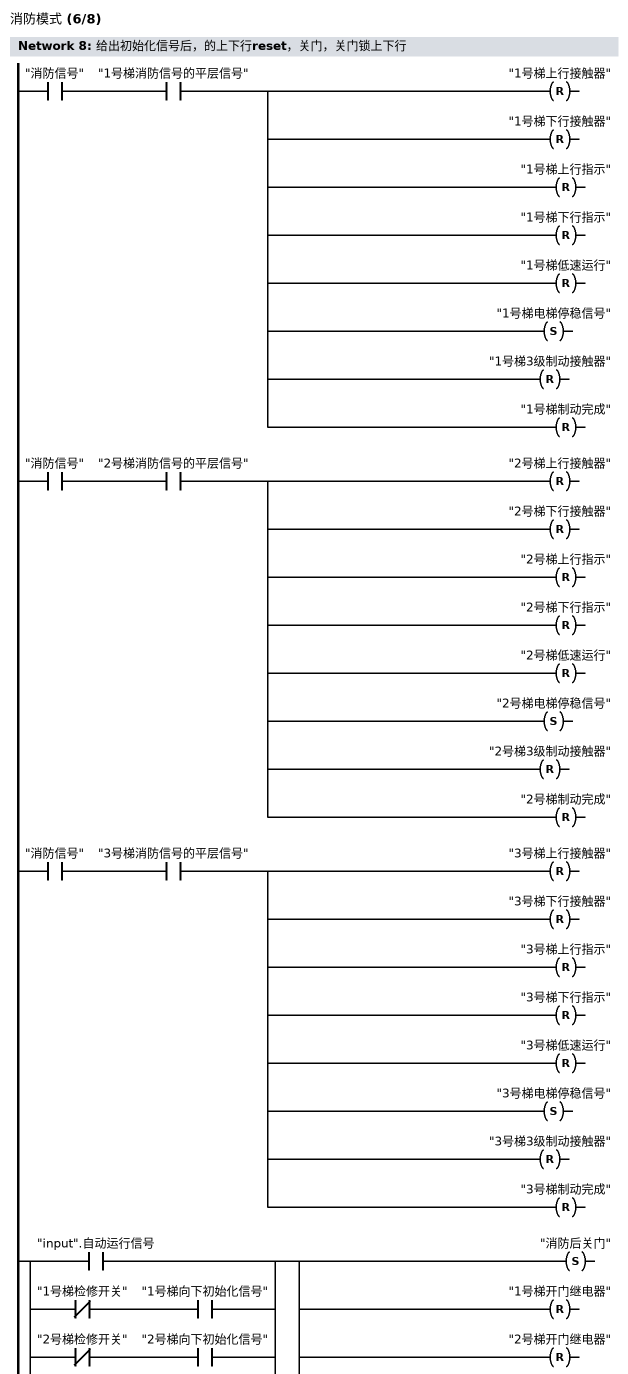
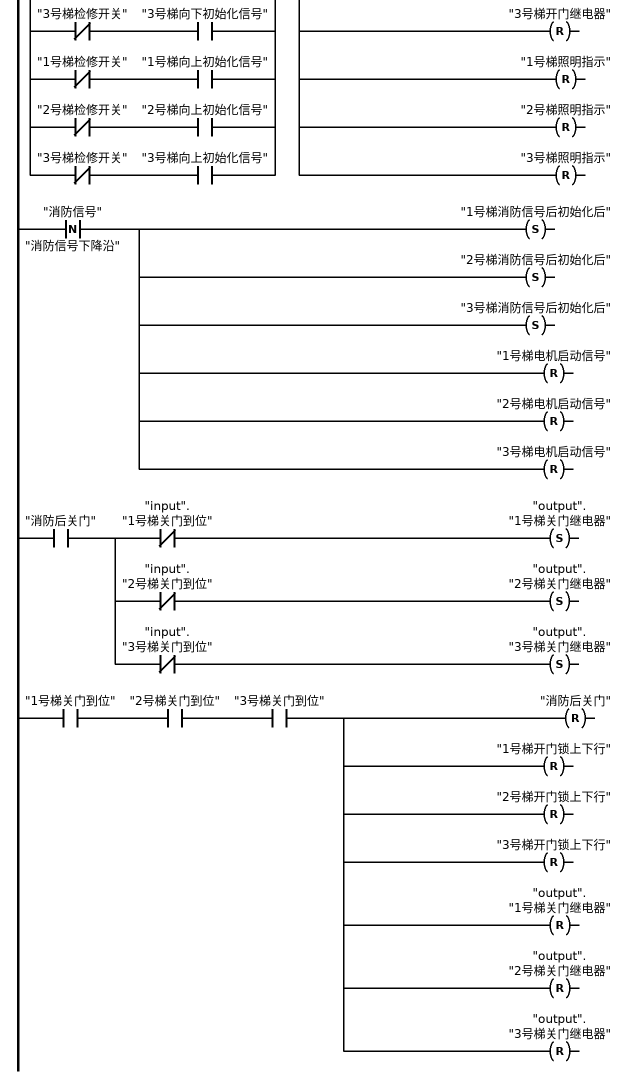
   RUNG wire#powerrail
      Contact( "消防信号" )
      Contact( "1号梯消防信号的平层信号" )
      wire#w1
      R_Coil( "1号梯上行接触器" )
   END_RUNG
   RUNG wire#w1
      R_Coil( "1号梯下行接触器" )
   END_RUNG
   RUNG wire#w1
      R_Coil( "1号梯上行指示" )
   END_RUNG
   RUNG wire#w1
      R_Coil( "1号梯下行指示" )
   END_RUNG
   RUNG wire#w1
      R_Coil( "1号梯低速运行" )
   END_RUNG
   RUNG wire#w1
      S_Coil( "1号梯电梯停稳信号" )
   END_RUNG
   RUNG wire#w1
      R_Coil( "1号梯3级制动接触器" )
   END_RUNG
   RUNG wire#w1
      R_Coil( "1号梯制动完成" )
   END_RUNG
   RUNG wire#powerrail
      Contact( "消防信号" )
      Contact( "2号梯消防信号的平层信号" )
      wire#w2
      R_Coil( "2号梯上行接触器" )
   END_RUNG
   RUNG wire#w2
      R_Coil( "2号梯下行接触器" )
   END_RUNG
   RUNG wire#w2
      R_Coil( "2号梯上行指示" )
   END_RUNG
   RUNG wire#w2
      R_Coil( "2号梯下行指示" )
   END_RUNG
   RUNG wire#w2
      R_Coil( "2号梯低速运行" )
   END_RUNG
   RUNG wire#w2
      S_Coil( "2号梯电梯停稳信号" )
   END_RUNG
   RUNG wire#w2
      R_Coil( "2号梯3级制动接触器" )
   END_RUNG
   RUNG wire#w2
      R_Coil( "2号梯制动完成" )
   END_RUNG
   RUNG wire#powerrail
      Contact( "消防信号" )
      Contact( "3号梯消防信号的平层信号" )
      wire#w3
      R_Coil( "3号梯上行接触器" )
   END_RUNG
   RUNG wire#w3
      R_Coil( "3号梯下行接触器" )
   END_RUNG
   RUNG wire#w3
      R_Coil( "3号梯上行指示" )
   END_RUNG
   RUNG wire#w3
      R_Coil( "3号梯下行指示" )
   END_RUNG
   RUNG wire#w3
      R_Coil( "3号梯低速运行" )
   END_RUNG
   RUNG wire#w3
      S_Coil( "3号梯电梯停稳信号" )
   END_RUNG
   RUNG wire#w3
      R_Coil( "3号梯3级制动接触器" )
   END_RUNG
   RUNG wire#w3
      R_Coil( "3号梯制动完成" )
   END_RUNG
   RUNG wire#powerrail
      Contact( "input".自动运行信号 )
      wire#w4
      S_Coil( "消防后关门" )
   END_RUNG
   RUNG wire#powerrail
      I_Contact( "1号梯检修开关" )
      Contact( "1号梯向下初始化信号" )
   END_RUNG wire#w4
   RUNG wire#powerrail
      I_Contact( "2号梯检修开关" )
      Contact( "2号梯向下初始化信号" )
   END_RUNG wire#w4
   RUNG wire#powerrail
      I_Contact( "3号梯检修开关" )
      Contact( "3号梯向下初始化信号" )
   END_RUNG wire#w4
   RUNG wire#powerrail
      I_Contact( "1号梯检修开关" )
      Contact( "1号梯向上初始化信号" )
   END_RUNG wire#w4
   RUNG wire#powerrail
      I_Contact( "2号梯检修开关" )
      Contact( "2号梯向上初始化信号" )
   END_RUNG wire#w4
   RUNG wire#powerrail
      I_Contact( "3号梯检修开关" )
      Contact( "3号梯向上初始化信号" )
   END_RUNG wire#w4
   RUNG wire#w4
      R_Coil( "1号梯开门继电器" )
   END_RUNG
   RUNG wire#w4
      R_Coil( "2号梯开门继电器" )
   END_RUNG
   RUNG wire#w4
      R_Coil( "3号梯开门继电器" )
   END_RUNG
   RUNG wire#w4
      R_Coil( "1号梯照明指示" )
   END_RUNG
   RUNG wire#w4
      R_Coil( "2号梯照明指示" )
   END_RUNG
   RUNG wire#w4
      R_Coil( "3号梯照明指示" )
   END_RUNG
   RUNG wire#powerrail
      N_Contact(operand := "消防信号", bit := "消防信号下降沿")
      wire#w5
      S_Coil( "1号梯消防信号后初始化后" )
   END_RUNG
   RUNG wire#w5
      S_Coil( "2号梯消防信号后初始化后" )
   END_RUNG
   RUNG wire#w5
      S_Coil( "3号梯消防信号后初始化后" )
   END_RUNG
   RUNG wire#w5
      R_Coil( "1号梯电机启动信号" )
   END_RUNG
   RUNG wire#w5
      R_Coil( "2号梯电机启动信号" )
   END_RUNG
   RUNG wire#w5
      R_Coil( "3号梯电机启动信号" )
   END_RUNG
   RUNG wire#powerrail
      Contact( "消防后关门" )
      wire#w6
      I_Contact( "input"."1号梯关门到位" )
      S_Coil( "output"."1号梯关门继电器" )
   END_RUNG
   RUNG wire#w6
      I_Contact( "input"."2号梯关门到位" )
      S_Coil( "output"."2号梯关门继电器" )
   END_RUNG
   RUNG wire#w6
      I_Contact( "input"."3号梯关门到位" )
      S_Coil( "output"."3号梯关门继电器" )
   END_RUNG
   RUNG wire#powerrail
      Contact( "1号梯关门到位" )
      Contact( "2号梯关门到位" )
      Contact( "3号梯关门到位" )
      wire#w7
      R_Coil( "消防后关门" )
   END_RUNG
   RUNG wire#w7
      R_Coil( "1号梯开门锁上下行" )
   END_RUNG
   RUNG wire#w7
      R_Coil( "2号梯开门锁上下行" )
   END_RUNG
   RUNG wire#w7
      R_Coil( "3号梯开门锁上下行" )
   END_RUNG
   RUNG wire#w7
      R_Coil( "output"."1号梯关门继电器" )
   END_RUNG
   RUNG wire#w7
      R_Coil( "output"."2号梯关门继电器" )
   END_RUNG
   RUNG wire#w7
      R_Coil( "output"."3号梯关门继电器" )
   END_RUNG
   // the same network as SCL:
   IF "消防信号" AND "1号梯消防信号的平层信号" THEN
       "1号梯上行接触器" := FALSE;
       "1号梯下行接触器" := FALSE;
       "1号梯上行指示" := FALSE;
       "1号梯下行指示" := FALSE;
       "1号梯低速运行" := FALSE;
       "1号梯电梯停稳信号" := TRUE;
       "1号梯3级制动接触器" := FALSE;
       "1号梯制动完成" := FALSE;
   END_IF;
   IF "消防信号" AND "2号梯消防信号的平层信号" THEN
       "2号梯上行接触器" := FALSE;
       "2号梯下行接触器" := FALSE;
       "2号梯上行指示" := FALSE;
       "2号梯下行指示" := FALSE;
       "2号梯低速运行" := FALSE;
       "2号梯电梯停稳信号" := TRUE;
       "2号梯3级制动接触器" := FALSE;
       "2号梯制动完成" := FALSE;
   END_IF;
   IF "消防信号" AND "3号梯消防信号的平层信号" THEN
       "3号梯上行接触器" := FALSE;
       "3号梯下行接触器" := FALSE;
       "3号梯上行指示" := FALSE;
       "3号梯下行指示" := FALSE;
       "3号梯低速运行" := FALSE;
       "3号梯电梯停稳信号" := TRUE;
       "3号梯3级制动接触器" := FALSE;
       "3号梯制动完成" := FALSE;
   END_IF;
   IF "input".自动运行信号 OR (NOT "1号梯检修开关" AND "1号梯向下初始化信号") OR (NOT "2号梯检修开关" AND "2号梯向下初始化信号") OR (NOT "3号梯检修开关" AND "3号梯向下初始化信号") OR (NOT "1号梯检修开关" AND "1号梯向上初始化信号") OR (NOT "2号梯检修开关" AND "2号梯向上初始化信号") OR (NOT "3号梯检修开关" AND "3号梯向上初始化信号") THEN
       "消防后关门" := TRUE;
       "1号梯开门继电器" := FALSE;
       "2号梯开门继电器" := FALSE;
       "3号梯开门继电器" := FALSE;
       "1号梯照明指示" := FALSE;
       "2号梯照明指示" := FALSE;
       "3号梯照明指示" := FALSE;
   END_IF;
   #_w1 := NOT "消防信号" AND "消防信号下降沿";   // falling edge of "消防信号"
   "消防信号下降沿" := "消防信号";
   IF #_w1 THEN
       "1号梯消防信号后初始化后" := TRUE;
       "2号梯消防信号后初始化后" := TRUE;
       "3号梯消防信号后初始化后" := TRUE;
       "1号梯电机启动信号" := FALSE;
       "2号梯电机启动信号" := FALSE;
       "3号梯电机启动信号" := FALSE;
   END_IF;
   IF "消防后关门" AND NOT "input"."1号梯关门到位" THEN "output"."1号梯关门继电器" := TRUE; END_IF;
   IF "消防后关门" AND NOT "input"."2号梯关门到位" THEN "output"."2号梯关门继电器" := TRUE; END_IF;
   IF "消防后关门" AND NOT "input"."3号梯关门到位" THEN "output"."3号梯关门继电器" := TRUE; END_IF;
   IF "1号梯关门到位" AND "2号梯关门到位" AND "3号梯关门到位" THEN
       "消防后关门" := FALSE;
       "1号梯开门锁上下行" := FALSE;
       "2号梯开门锁上下行" := FALSE;
       "3号梯开门锁上下行" := FALSE;
       "output"."1号梯关门继电器" := FALSE;
       "output"."2号梯关门继电器" := FALSE;
       "output"."3号梯关门继电器" := FALSE;
   END_IF;
END_REGION

REGION Network 9: 群控输入的reset的reset
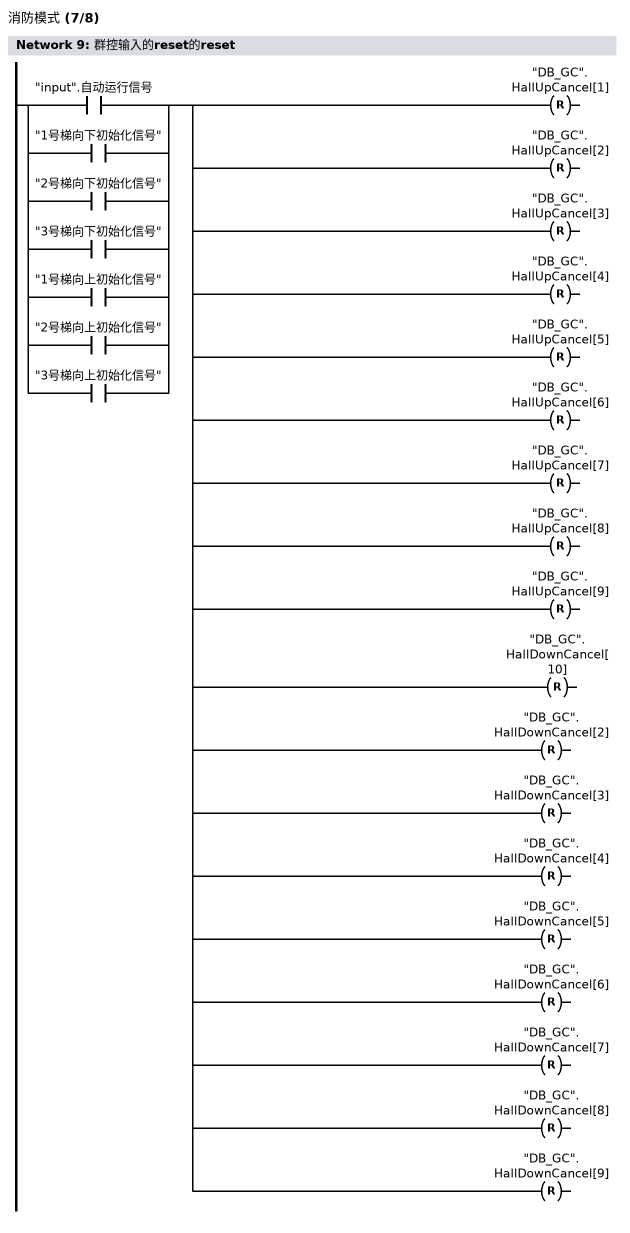
   RUNG wire#powerrail
      Contact( "input".自动运行信号 )
      wire#w1
      R_Coil( "DB_GC".HallUpCancel[1] )
   END_RUNG
   RUNG wire#powerrail
      Contact( "1号梯向下初始化信号" )
   END_RUNG wire#w1
   RUNG wire#powerrail
      Contact( "2号梯向下初始化信号" )
   END_RUNG wire#w1
   RUNG wire#powerrail
      Contact( "3号梯向下初始化信号" )
   END_RUNG wire#w1
   RUNG wire#powerrail
      Contact( "1号梯向上初始化信号" )
   END_RUNG wire#w1
   RUNG wire#powerrail
      Contact( "2号梯向上初始化信号" )
   END_RUNG wire#w1
   RUNG wire#powerrail
      Contact( "3号梯向上初始化信号" )
   END_RUNG wire#w1
   RUNG wire#w1
      R_Coil( "DB_GC".HallUpCancel[2] )
   END_RUNG
   RUNG wire#w1
      R_Coil( "DB_GC".HallUpCancel[3] )
   END_RUNG
   RUNG wire#w1
      R_Coil( "DB_GC".HallUpCancel[4] )
   END_RUNG
   RUNG wire#w1
      R_Coil( "DB_GC".HallUpCancel[5] )
   END_RUNG
   RUNG wire#w1
      R_Coil( "DB_GC".HallUpCancel[6] )
   END_RUNG
   RUNG wire#w1
      R_Coil( "DB_GC".HallUpCancel[7] )
   END_RUNG
   RUNG wire#w1
      R_Coil( "DB_GC".HallUpCancel[8] )
   END_RUNG
   RUNG wire#w1
      R_Coil( "DB_GC".HallUpCancel[9] )
   END_RUNG
   RUNG wire#w1
      R_Coil( "DB_GC".HallDownCancel[10] )
   END_RUNG
   RUNG wire#w1
      R_Coil( "DB_GC".HallDownCancel[2] )
   END_RUNG
   RUNG wire#w1
      R_Coil( "DB_GC".HallDownCancel[3] )
   END_RUNG
   RUNG wire#w1
      R_Coil( "DB_GC".HallDownCancel[4] )
   END_RUNG
   RUNG wire#w1
      R_Coil( "DB_GC".HallDownCancel[5] )
   END_RUNG
   RUNG wire#w1
      R_Coil( "DB_GC".HallDownCancel[6] )
   END_RUNG
   RUNG wire#w1
      R_Coil( "DB_GC".HallDownCancel[7] )
   END_RUNG
   RUNG wire#w1
      R_Coil( "DB_GC".HallDownCancel[8] )
   END_RUNG
   RUNG wire#w1
      R_Coil( "DB_GC".HallDownCancel[9] )
   END_RUNG
   // the same network as SCL:
   IF "input".自动运行信号 OR "1号梯向下初始化信号" OR "2号梯向下初始化信号" OR "3号梯向下初始化信号" OR "1号梯向上初始化信号" OR "2号梯向上初始化信号" OR "3号梯向上初始化信号" THEN
       "DB_GC".HallUpCancel[1] := FALSE;
       "DB_GC".HallUpCancel[2] := FALSE;
       "DB_GC".HallUpCancel[3] := FALSE;
       "DB_GC".HallUpCancel[4] := FALSE;
       "DB_GC".HallUpCancel[5] := FALSE;
       "DB_GC".HallUpCancel[6] := FALSE;
       "DB_GC".HallUpCancel[7] := FALSE;
       "DB_GC".HallUpCancel[8] := FALSE;
       "DB_GC".HallUpCancel[9] := FALSE;
       "DB_GC".HallDownCancel[10] := FALSE;
       "DB_GC".HallDownCancel[2] := FALSE;
       "DB_GC".HallDownCancel[3] := FALSE;
       "DB_GC".HallDownCancel[4] := FALSE;
       "DB_GC".HallDownCancel[5] := FALSE;
       "DB_GC".HallDownCancel[6] := FALSE;
       "DB_GC".HallDownCancel[7] := FALSE;
       "DB_GC".HallDownCancel[8] := FALSE;
       "DB_GC".HallDownCancel[9] := FALSE;
   END_IF;
END_REGION

REGION Network 10: 第二次自动运行信号
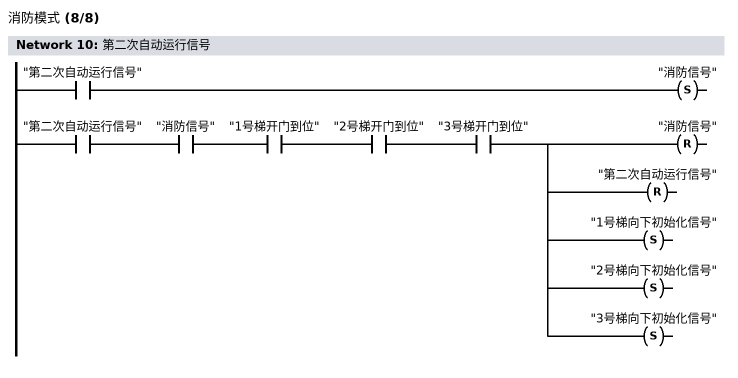
   RUNG wire#powerrail
      Contact( "第二次自动运行信号" )
      S_Coil( "消防信号" )
   END_RUNG
   RUNG wire#powerrail
      Contact( "第二次自动运行信号" )
      Contact( "消防信号" )
      Contact( "1号梯开门到位" )
      Contact( "2号梯开门到位" )
      Contact( "3号梯开门到位" )
      wire#w1
      R_Coil( "消防信号" )
   END_RUNG
   RUNG wire#w1
      R_Coil( "第二次自动运行信号" )
   END_RUNG
   RUNG wire#w1
      S_Coil( "1号梯向下初始化信号" )
   END_RUNG
   RUNG wire#w1
      S_Coil( "2号梯向下初始化信号" )
   END_RUNG
   RUNG wire#w1
      S_Coil( "3号梯向下初始化信号" )
   END_RUNG
   // the same network as SCL:
   IF "第二次自动运行信号" THEN "消防信号" := TRUE; END_IF;
   #_w1 := "第二次自动运行信号" AND "消防信号" AND "1号梯开门到位" AND "2号梯开门到位" AND "3号梯开门到位";
   IF #_w1 THEN
       "消防信号" := FALSE;
       "第二次自动运行信号" := FALSE;
       "1号梯向下初始化信号" := TRUE;
       "2号梯向下初始化信号" := TRUE;
       "3号梯向下初始化信号" := TRUE;
   END_IF;
END_REGION
END_FUNCTION

FUNCTION "1号电梯初始化" : Void   // FC7, LAD
{ S7_Optimized_Access := 'TRUE' }
VERSION : 0.1
   VAR_TEMP   // added for the SCL form of the ladder/FBD networks
      _w1 : Bool;
   END_VAR
BEGIN

REGION Network 1: 上下行初始化选择
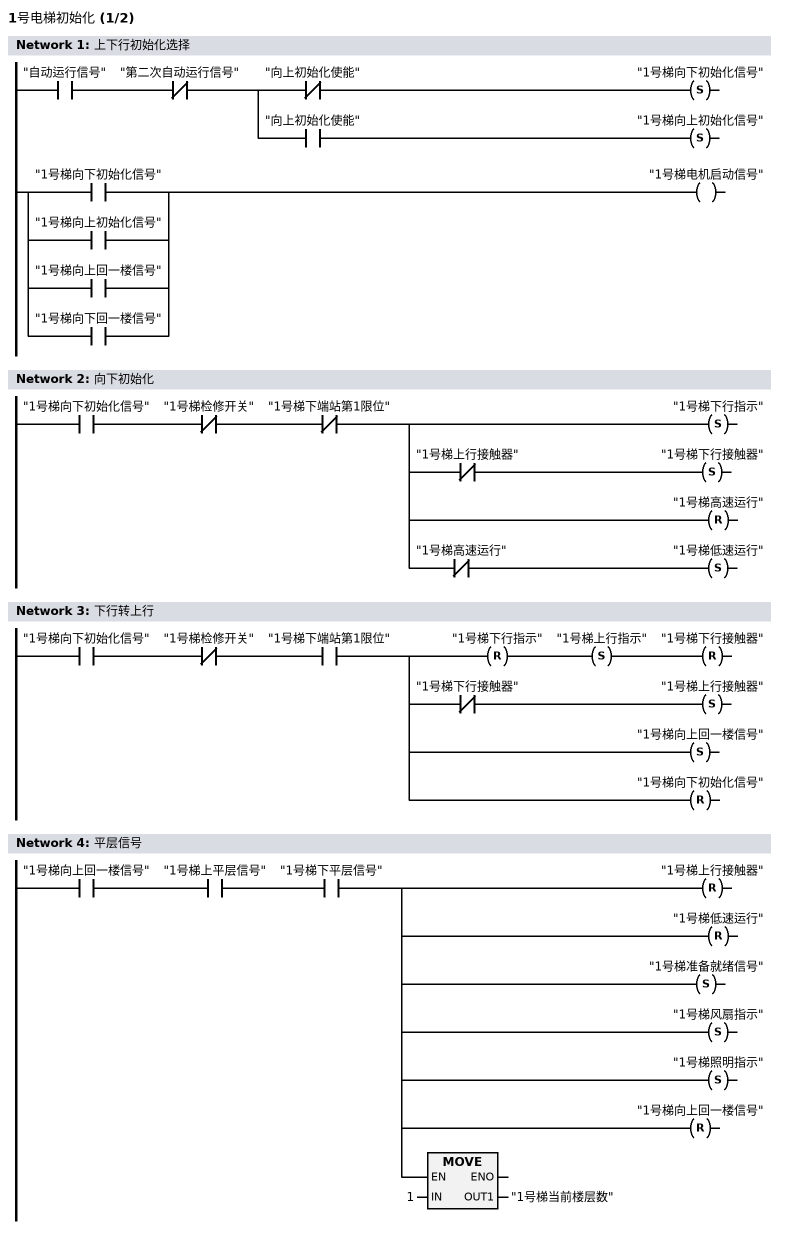
   RUNG wire#powerrail
      Contact( "自动运行信号" )
      I_Contact( "第二次自动运行信号" )
      wire#w1
      I_Contact( "向上初始化使能" )
      S_Coil( "1号梯向下初始化信号" )
   END_RUNG
   RUNG wire#w1
      Contact( "向上初始化使能" )
      S_Coil( "1号梯向上初始化信号" )
   END_RUNG
   RUNG wire#powerrail
      Contact( "1号梯向下初始化信号" )
      wire#w2
      Coil( "1号梯电机启动信号" )
   END_RUNG
   RUNG wire#powerrail
      Contact( "1号梯向上初始化信号" )
   END_RUNG wire#w2
   RUNG wire#powerrail
      Contact( "1号梯向上回一楼信号" )
   END_RUNG wire#w2
   RUNG wire#powerrail
      Contact( "1号梯向下回一楼信号" )
   END_RUNG wire#w2
   // the same network as SCL:
   #_w1 := "自动运行信号" AND NOT "第二次自动运行信号";
   IF #_w1 AND NOT "向上初始化使能" THEN "1号梯向下初始化信号" := TRUE; END_IF;
   IF #_w1 AND "向上初始化使能" THEN "1号梯向上初始化信号" := TRUE; END_IF;
   "1号梯电机启动信号" := "1号梯向下初始化信号" OR "1号梯向上初始化信号" OR "1号梯向上回一楼信号" OR "1号梯向下回一楼信号";
END_REGION

REGION Network 2: 向下初始化
   RUNG wire#powerrail
      Contact( "1号梯向下初始化信号" )
      I_Contact( "1号梯检修开关" )
      I_Contact( "1号梯下端站第1限位" )
      wire#w1
      S_Coil( "1号梯下行指示" )
   END_RUNG
   RUNG wire#w1
      I_Contact( "1号梯上行接触器" )
      S_Coil( "1号梯下行接触器" )
   END_RUNG
   RUNG wire#w1
      R_Coil( "1号梯高速运行" )
   END_RUNG
   RUNG wire#w1
      I_Contact( "1号梯高速运行" )
      S_Coil( "1号梯低速运行" )
   END_RUNG
   // the same network as SCL:
   #_w1 := "1号梯向下初始化信号" AND NOT "1号梯检修开关" AND NOT "1号梯下端站第1限位";
   IF #_w1 THEN "1号梯下行指示" := TRUE; END_IF;
   IF #_w1 AND NOT "1号梯上行接触器" THEN "1号梯下行接触器" := TRUE; END_IF;
   IF #_w1 THEN "1号梯高速运行" := FALSE; END_IF;
   IF #_w1 AND NOT "1号梯高速运行" THEN "1号梯低速运行" := TRUE; END_IF;
END_REGION

REGION Network 3: 下行转上行
   RUNG wire#powerrail
      Contact( "1号梯向下初始化信号" )
      I_Contact( "1号梯检修开关" )
      Contact( "1号梯下端站第1限位" )
      wire#w1
      R_Coil( "1号梯下行指示" )
      S_Coil( "1号梯上行指示" )
      R_Coil( "1号梯下行接触器" )
   END_RUNG
   RUNG wire#w1
      I_Contact( "1号梯下行接触器" )
      S_Coil( "1号梯上行接触器" )
   END_RUNG
   RUNG wire#w1
      S_Coil( "1号梯向上回一楼信号" )
   END_RUNG
   RUNG wire#w1
      R_Coil( "1号梯向下初始化信号" )
   END_RUNG
   // the same network as SCL:
   #_w1 := "1号梯向下初始化信号" AND NOT "1号梯检修开关" AND "1号梯下端站第1限位";
   IF #_w1 THEN
       "1号梯下行指示" := FALSE;
       "1号梯上行指示" := TRUE;
       "1号梯下行接触器" := FALSE;
   END_IF;
   IF #_w1 AND NOT "1号梯下行接触器" THEN "1号梯上行接触器" := TRUE; END_IF;
   IF #_w1 THEN
       "1号梯向上回一楼信号" := TRUE;
       "1号梯向下初始化信号" := FALSE;
   END_IF;
END_REGION

REGION Network 4: 平层信号
   RUNG wire#powerrail
      Contact( "1号梯向上回一楼信号" )
      Contact( "1号梯上平层信号" )
      Contact( "1号梯下平层信号" )
      wire#w1
      R_Coil( "1号梯上行接触器" )
   END_RUNG
   RUNG wire#w1
      R_Coil( "1号梯低速运行" )
   END_RUNG
   RUNG wire#w1
      S_Coil( "1号梯准备就绪信号" )
   END_RUNG
   RUNG wire#w1
      S_Coil( "1号梯风扇指示" )
   END_RUNG
   RUNG wire#w1
      S_Coil( "1号梯照明指示" )
   END_RUNG
   RUNG wire#w1
      R_Coil( "1号梯向上回一楼信号" )
   END_RUNG
   RUNG wire#w1
      Move(in := 1, out1 => "1号梯当前楼层数")
   END_RUNG
   // the same network as SCL:
   IF "1号梯向上回一楼信号" AND "1号梯上平层信号" AND "1号梯下平层信号" THEN
       "1号梯上行接触器" := FALSE;
       "1号梯低速运行" := FALSE;
       "1号梯准备就绪信号" := TRUE;
       "1号梯风扇指示" := TRUE;
       "1号梯照明指示" := TRUE;
   END_IF;
   #_w1 := "1号梯向上回一楼信号" AND "1号梯上平层信号" AND "1号梯下平层信号";
   IF #_w1 THEN
       "1号梯向上回一楼信号" := FALSE;
       "1号梯当前楼层数" := 1;
   END_IF;
END_REGION

REGION Network 5: 向上初始化
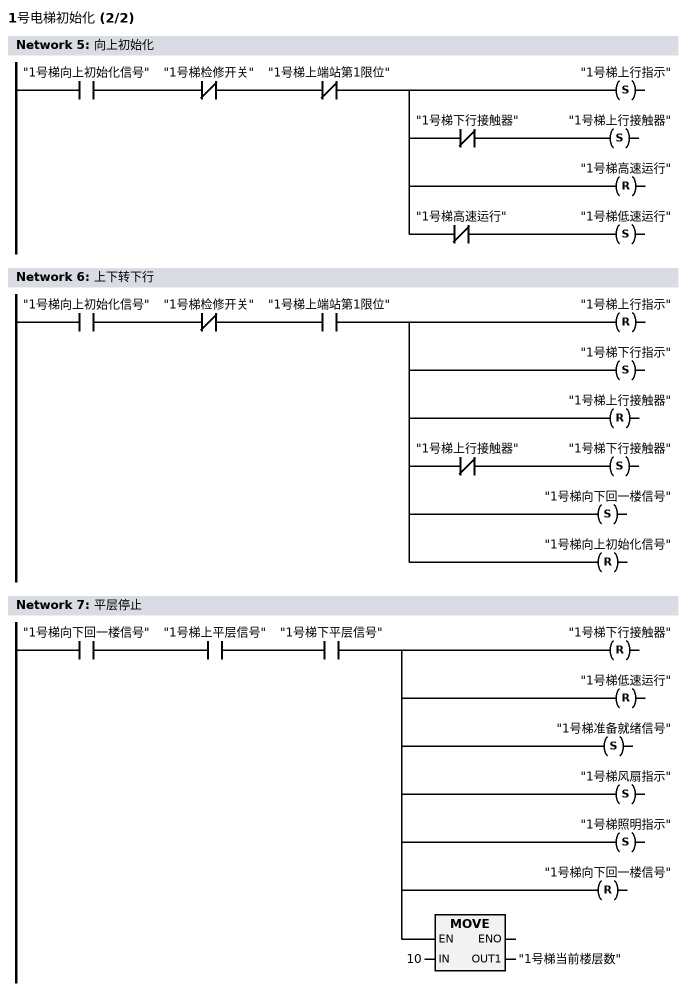
   RUNG wire#powerrail
      Contact( "1号梯向上初始化信号" )
      I_Contact( "1号梯检修开关" )
      I_Contact( "1号梯上端站第1限位" )
      wire#w1
      S_Coil( "1号梯上行指示" )
   END_RUNG
   RUNG wire#w1
      I_Contact( "1号梯下行接触器" )
      S_Coil( "1号梯上行接触器" )
   END_RUNG
   RUNG wire#w1
      R_Coil( "1号梯高速运行" )
   END_RUNG
   RUNG wire#w1
      I_Contact( "1号梯高速运行" )
      S_Coil( "1号梯低速运行" )
   END_RUNG
   // the same network as SCL:
   #_w1 := "1号梯向上初始化信号" AND NOT "1号梯检修开关" AND NOT "1号梯上端站第1限位";
   IF #_w1 THEN "1号梯上行指示" := TRUE; END_IF;
   IF #_w1 AND NOT "1号梯下行接触器" THEN "1号梯上行接触器" := TRUE; END_IF;
   IF #_w1 THEN "1号梯高速运行" := FALSE; END_IF;
   IF #_w1 AND NOT "1号梯高速运行" THEN "1号梯低速运行" := TRUE; END_IF;
END_REGION

REGION Network 6: 上下转下行
   RUNG wire#powerrail
      Contact( "1号梯向上初始化信号" )
      I_Contact( "1号梯检修开关" )
      Contact( "1号梯上端站第1限位" )
      wire#w1
      R_Coil( "1号梯上行指示" )
   END_RUNG
   RUNG wire#w1
      S_Coil( "1号梯下行指示" )
   END_RUNG
   RUNG wire#w1
      R_Coil( "1号梯上行接触器" )
   END_RUNG
   RUNG wire#w1
      I_Contact( "1号梯上行接触器" )
      S_Coil( "1号梯下行接触器" )
   END_RUNG
   RUNG wire#w1
      S_Coil( "1号梯向下回一楼信号" )
   END_RUNG
   RUNG wire#w1
      R_Coil( "1号梯向上初始化信号" )
   END_RUNG
   // the same network as SCL:
   #_w1 := "1号梯向上初始化信号" AND NOT "1号梯检修开关" AND "1号梯上端站第1限位";
   IF #_w1 THEN
       "1号梯上行指示" := FALSE;
       "1号梯下行指示" := TRUE;
       "1号梯上行接触器" := FALSE;
   END_IF;
   IF #_w1 AND NOT "1号梯上行接触器" THEN "1号梯下行接触器" := TRUE; END_IF;
   IF #_w1 THEN
       "1号梯向下回一楼信号" := TRUE;
       "1号梯向上初始化信号" := FALSE;
   END_IF;
END_REGION

REGION Network 7: 平层停止
   RUNG wire#powerrail
      Contact( "1号梯向下回一楼信号" )
      Contact( "1号梯上平层信号" )
      Contact( "1号梯下平层信号" )
      wire#w1
      R_Coil( "1号梯下行接触器" )
   END_RUNG
   RUNG wire#w1
      R_Coil( "1号梯低速运行" )
   END_RUNG
   RUNG wire#w1
      S_Coil( "1号梯准备就绪信号" )
   END_RUNG
   RUNG wire#w1
      S_Coil( "1号梯风扇指示" )
   END_RUNG
   RUNG wire#w1
      S_Coil( "1号梯照明指示" )
   END_RUNG
   RUNG wire#w1
      R_Coil( "1号梯向下回一楼信号" )
   END_RUNG
   RUNG wire#w1
      Move(in := 10, out1 => "1号梯当前楼层数")
   END_RUNG
   // the same network as SCL:
   IF "1号梯向下回一楼信号" AND "1号梯上平层信号" AND "1号梯下平层信号" THEN
       "1号梯下行接触器" := FALSE;
       "1号梯低速运行" := FALSE;
       "1号梯准备就绪信号" := TRUE;
       "1号梯风扇指示" := TRUE;
       "1号梯照明指示" := TRUE;
   END_IF;
   #_w1 := "1号梯向下回一楼信号" AND "1号梯上平层信号" AND "1号梯下平层信号";
   IF #_w1 THEN
       "1号梯向下回一楼信号" := FALSE;
       "1号梯当前楼层数" := 10;
   END_IF;
END_REGION
END_FUNCTION

FUNCTION "2号电梯初始化" : Void   // FC8, LAD
{ S7_Optimized_Access := 'TRUE' }
VERSION : 0.1
   VAR_TEMP   // added for the SCL form of the ladder/FBD networks
      _w1 : Bool;
   END_VAR
BEGIN

REGION Network 1: 上下行初始化选择
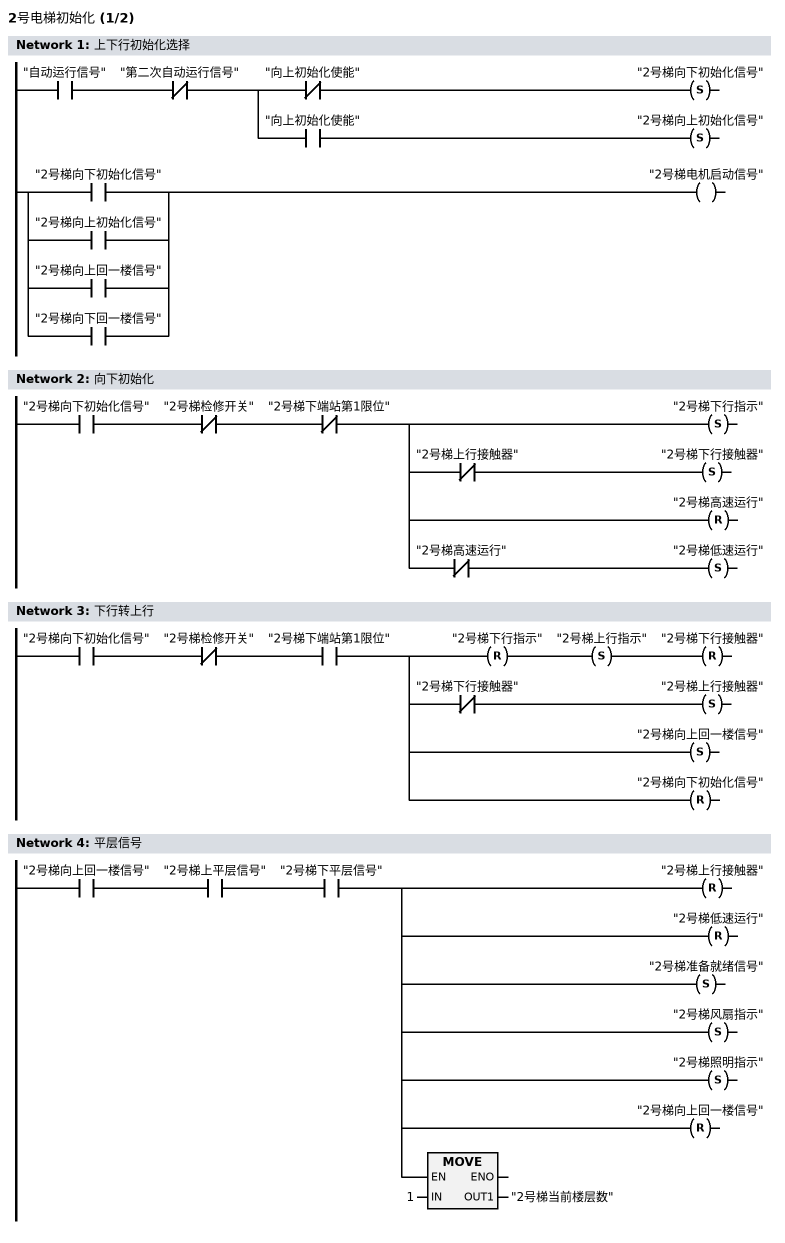
   RUNG wire#powerrail
      Contact( "自动运行信号" )
      I_Contact( "第二次自动运行信号" )
      wire#w1
      I_Contact( "向上初始化使能" )
      S_Coil( "2号梯向下初始化信号" )
   END_RUNG
   RUNG wire#w1
      Contact( "向上初始化使能" )
      S_Coil( "2号梯向上初始化信号" )
   END_RUNG
   RUNG wire#powerrail
      Contact( "2号梯向下初始化信号" )
      wire#w2
      Coil( "2号梯电机启动信号" )
   END_RUNG
   RUNG wire#powerrail
      Contact( "2号梯向上初始化信号" )
   END_RUNG wire#w2
   RUNG wire#powerrail
      Contact( "2号梯向上回一楼信号" )
   END_RUNG wire#w2
   RUNG wire#powerrail
      Contact( "2号梯向下回一楼信号" )
   END_RUNG wire#w2
   // the same network as SCL:
   #_w1 := "自动运行信号" AND NOT "第二次自动运行信号";
   IF #_w1 AND NOT "向上初始化使能" THEN "2号梯向下初始化信号" := TRUE; END_IF;
   IF #_w1 AND "向上初始化使能" THEN "2号梯向上初始化信号" := TRUE; END_IF;
   "2号梯电机启动信号" := "2号梯向下初始化信号" OR "2号梯向上初始化信号" OR "2号梯向上回一楼信号" OR "2号梯向下回一楼信号";
END_REGION

REGION Network 2: 向下初始化
   RUNG wire#powerrail
      Contact( "2号梯向下初始化信号" )
      I_Contact( "2号梯检修开关" )
      I_Contact( "2号梯下端站第1限位" )
      wire#w1
      S_Coil( "2号梯下行指示" )
   END_RUNG
   RUNG wire#w1
      I_Contact( "2号梯上行接触器" )
      S_Coil( "2号梯下行接触器" )
   END_RUNG
   RUNG wire#w1
      R_Coil( "2号梯高速运行" )
   END_RUNG
   RUNG wire#w1
      I_Contact( "2号梯高速运行" )
      S_Coil( "2号梯低速运行" )
   END_RUNG
   // the same network as SCL:
   #_w1 := "2号梯向下初始化信号" AND NOT "2号梯检修开关" AND NOT "2号梯下端站第1限位";
   IF #_w1 THEN "2号梯下行指示" := TRUE; END_IF;
   IF #_w1 AND NOT "2号梯上行接触器" THEN "2号梯下行接触器" := TRUE; END_IF;
   IF #_w1 THEN "2号梯高速运行" := FALSE; END_IF;
   IF #_w1 AND NOT "2号梯高速运行" THEN "2号梯低速运行" := TRUE; END_IF;
END_REGION

REGION Network 3: 下行转上行
   RUNG wire#powerrail
      Contact( "2号梯向下初始化信号" )
      I_Contact( "2号梯检修开关" )
      Contact( "2号梯下端站第1限位" )
      wire#w1
      R_Coil( "2号梯下行指示" )
      S_Coil( "2号梯上行指示" )
      R_Coil( "2号梯下行接触器" )
   END_RUNG
   RUNG wire#w1
      I_Contact( "2号梯下行接触器" )
      S_Coil( "2号梯上行接触器" )
   END_RUNG
   RUNG wire#w1
      S_Coil( "2号梯向上回一楼信号" )
   END_RUNG
   RUNG wire#w1
      R_Coil( "2号梯向下初始化信号" )
   END_RUNG
   // the same network as SCL:
   #_w1 := "2号梯向下初始化信号" AND NOT "2号梯检修开关" AND "2号梯下端站第1限位";
   IF #_w1 THEN
       "2号梯下行指示" := FALSE;
       "2号梯上行指示" := TRUE;
       "2号梯下行接触器" := FALSE;
   END_IF;
   IF #_w1 AND NOT "2号梯下行接触器" THEN "2号梯上行接触器" := TRUE; END_IF;
   IF #_w1 THEN
       "2号梯向上回一楼信号" := TRUE;
       "2号梯向下初始化信号" := FALSE;
   END_IF;
END_REGION

REGION Network 4: 平层信号
   RUNG wire#powerrail
      Contact( "2号梯向上回一楼信号" )
      Contact( "2号梯上平层信号" )
      Contact( "2号梯下平层信号" )
      wire#w1
      R_Coil( "2号梯上行接触器" )
   END_RUNG
   RUNG wire#w1
      R_Coil( "2号梯低速运行" )
   END_RUNG
   RUNG wire#w1
      S_Coil( "2号梯准备就绪信号" )
   END_RUNG
   RUNG wire#w1
      S_Coil( "2号梯风扇指示" )
   END_RUNG
   RUNG wire#w1
      S_Coil( "2号梯照明指示" )
   END_RUNG
   RUNG wire#w1
      R_Coil( "2号梯向上回一楼信号" )
   END_RUNG
   RUNG wire#w1
      Move(in := 1, out1 => "2号梯当前楼层数")
   END_RUNG
   // the same network as SCL:
   IF "2号梯向上回一楼信号" AND "2号梯上平层信号" AND "2号梯下平层信号" THEN
       "2号梯上行接触器" := FALSE;
       "2号梯低速运行" := FALSE;
       "2号梯准备就绪信号" := TRUE;
       "2号梯风扇指示" := TRUE;
       "2号梯照明指示" := TRUE;
   END_IF;
   #_w1 := "2号梯向上回一楼信号" AND "2号梯上平层信号" AND "2号梯下平层信号";
   IF #_w1 THEN
       "2号梯向上回一楼信号" := FALSE;
       "2号梯当前楼层数" := 1;
   END_IF;
END_REGION

REGION Network 5: 向上初始化
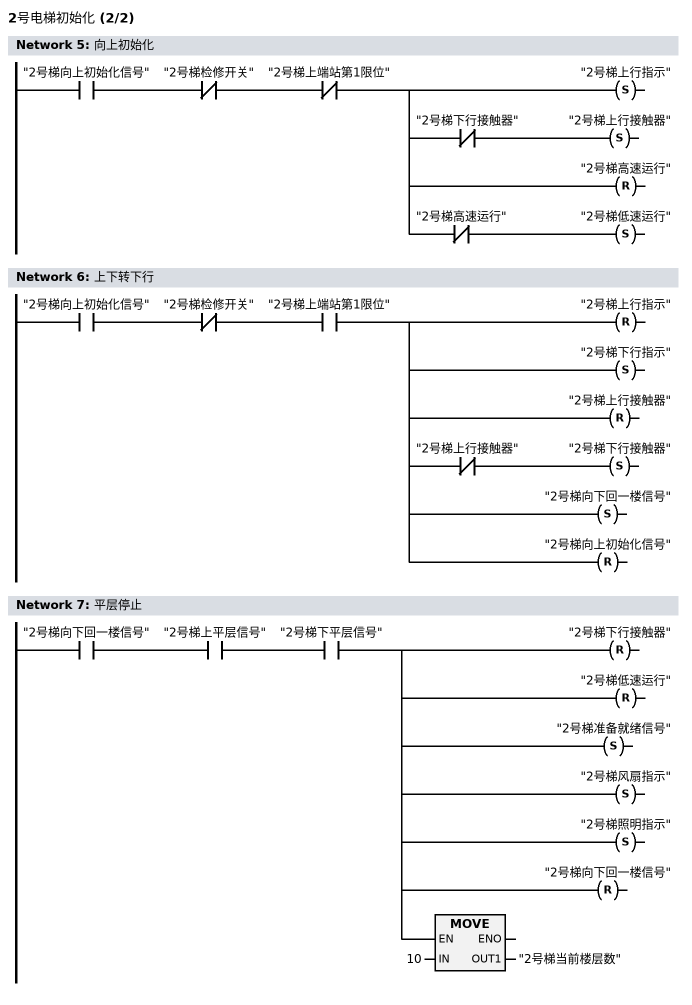
   RUNG wire#powerrail
      Contact( "2号梯向上初始化信号" )
      I_Contact( "2号梯检修开关" )
      I_Contact( "2号梯上端站第1限位" )
      wire#w1
      S_Coil( "2号梯上行指示" )
   END_RUNG
   RUNG wire#w1
      I_Contact( "2号梯下行接触器" )
      S_Coil( "2号梯上行接触器" )
   END_RUNG
   RUNG wire#w1
      R_Coil( "2号梯高速运行" )
   END_RUNG
   RUNG wire#w1
      I_Contact( "2号梯高速运行" )
      S_Coil( "2号梯低速运行" )
   END_RUNG
   // the same network as SCL:
   #_w1 := "2号梯向上初始化信号" AND NOT "2号梯检修开关" AND NOT "2号梯上端站第1限位";
   IF #_w1 THEN "2号梯上行指示" := TRUE; END_IF;
   IF #_w1 AND NOT "2号梯下行接触器" THEN "2号梯上行接触器" := TRUE; END_IF;
   IF #_w1 THEN "2号梯高速运行" := FALSE; END_IF;
   IF #_w1 AND NOT "2号梯高速运行" THEN "2号梯低速运行" := TRUE; END_IF;
END_REGION

REGION Network 6: 上下转下行
   RUNG wire#powerrail
      Contact( "2号梯向上初始化信号" )
      I_Contact( "2号梯检修开关" )
      Contact( "2号梯上端站第1限位" )
      wire#w1
      R_Coil( "2号梯上行指示" )
   END_RUNG
   RUNG wire#w1
      S_Coil( "2号梯下行指示" )
   END_RUNG
   RUNG wire#w1
      R_Coil( "2号梯上行接触器" )
   END_RUNG
   RUNG wire#w1
      I_Contact( "2号梯上行接触器" )
      S_Coil( "2号梯下行接触器" )
   END_RUNG
   RUNG wire#w1
      S_Coil( "2号梯向下回一楼信号" )
   END_RUNG
   RUNG wire#w1
      R_Coil( "2号梯向上初始化信号" )
   END_RUNG
   // the same network as SCL:
   #_w1 := "2号梯向上初始化信号" AND NOT "2号梯检修开关" AND "2号梯上端站第1限位";
   IF #_w1 THEN
       "2号梯上行指示" := FALSE;
       "2号梯下行指示" := TRUE;
       "2号梯上行接触器" := FALSE;
   END_IF;
   IF #_w1 AND NOT "2号梯上行接触器" THEN "2号梯下行接触器" := TRUE; END_IF;
   IF #_w1 THEN
       "2号梯向下回一楼信号" := TRUE;
       "2号梯向上初始化信号" := FALSE;
   END_IF;
END_REGION

REGION Network 7: 平层停止
   RUNG wire#powerrail
      Contact( "2号梯向下回一楼信号" )
      Contact( "2号梯上平层信号" )
      Contact( "2号梯下平层信号" )
      wire#w1
      R_Coil( "2号梯下行接触器" )
   END_RUNG
   RUNG wire#w1
      R_Coil( "2号梯低速运行" )
   END_RUNG
   RUNG wire#w1
      S_Coil( "2号梯准备就绪信号" )
   END_RUNG
   RUNG wire#w1
      S_Coil( "2号梯风扇指示" )
   END_RUNG
   RUNG wire#w1
      S_Coil( "2号梯照明指示" )
   END_RUNG
   RUNG wire#w1
      R_Coil( "2号梯向下回一楼信号" )
   END_RUNG
   RUNG wire#w1
      Move(in := 10, out1 => "2号梯当前楼层数")
   END_RUNG
   // the same network as SCL:
   IF "2号梯向下回一楼信号" AND "2号梯上平层信号" AND "2号梯下平层信号" THEN
       "2号梯下行接触器" := FALSE;
       "2号梯低速运行" := FALSE;
       "2号梯准备就绪信号" := TRUE;
       "2号梯风扇指示" := TRUE;
       "2号梯照明指示" := TRUE;
   END_IF;
   #_w1 := "2号梯向下回一楼信号" AND "2号梯上平层信号" AND "2号梯下平层信号";
   IF #_w1 THEN
       "2号梯向下回一楼信号" := FALSE;
       "2号梯当前楼层数" := 10;
   END_IF;
END_REGION
END_FUNCTION

FUNCTION "1号梯数码管显示" : Void   // FC9, LAD
{ S7_Optimized_Access := 'TRUE' }
VERSION : 0.1
   VAR_TEMP   // added for the SCL form of the ladder/FBD networks
      _w1 : Bool;
      _w2 : Bool;
      _w3 : Bool;
      _w4 : Bool;
      _w5 : Bool;
      _w6 : Bool;
      _w7 : Bool;
      _w8 : Bool;
      _w9 : Bool;
      _w10 : Bool;
      _w11 : Bool;
      _w12 : Bool;
      _w13 : Bool;
      _w14 : Bool;
      _w15 : Bool;
      _w16 : Bool;
      _w17 : Bool;
      _w18 : Bool;
      _w19 : Bool;
      _w20 : Bool;
   END_VAR
BEGIN

REGION Network 1: 根据楼层显示数码管
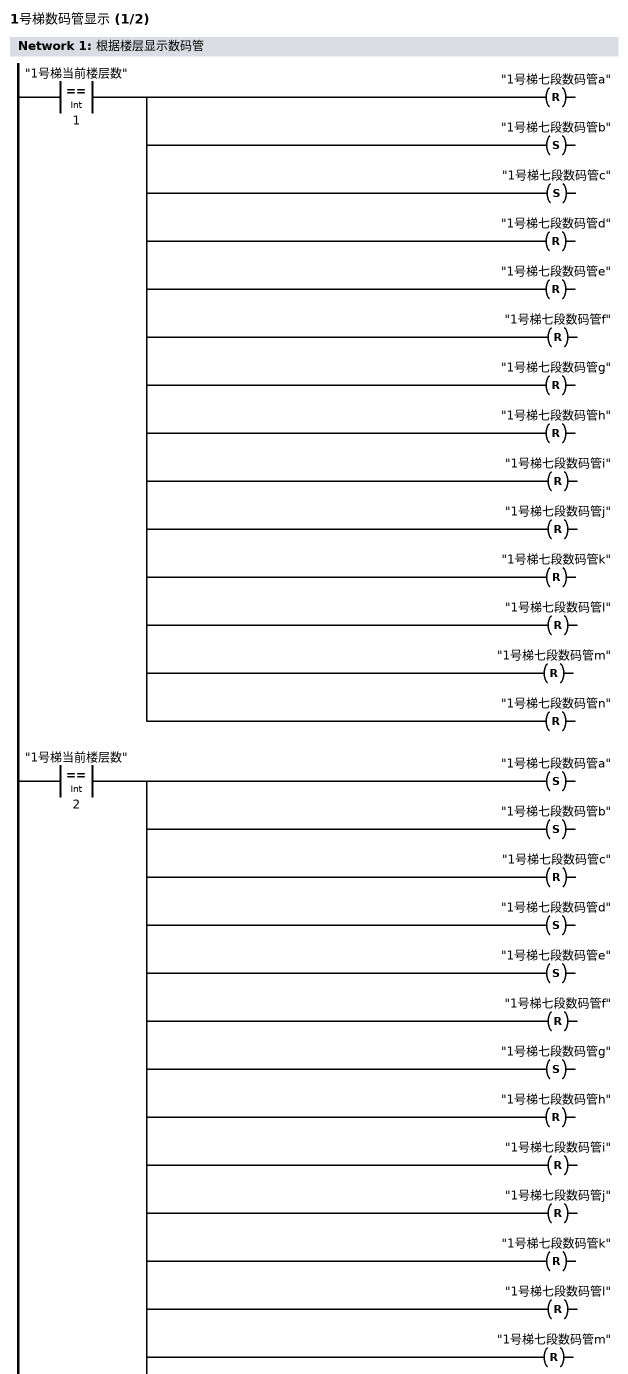
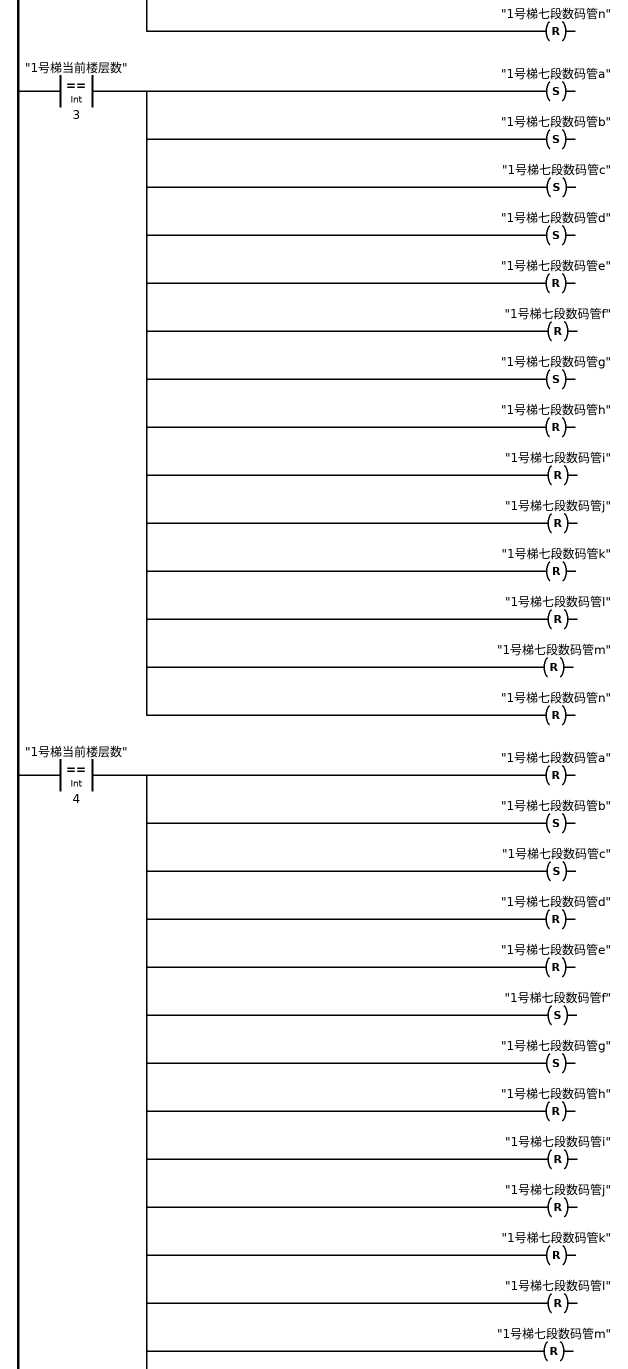
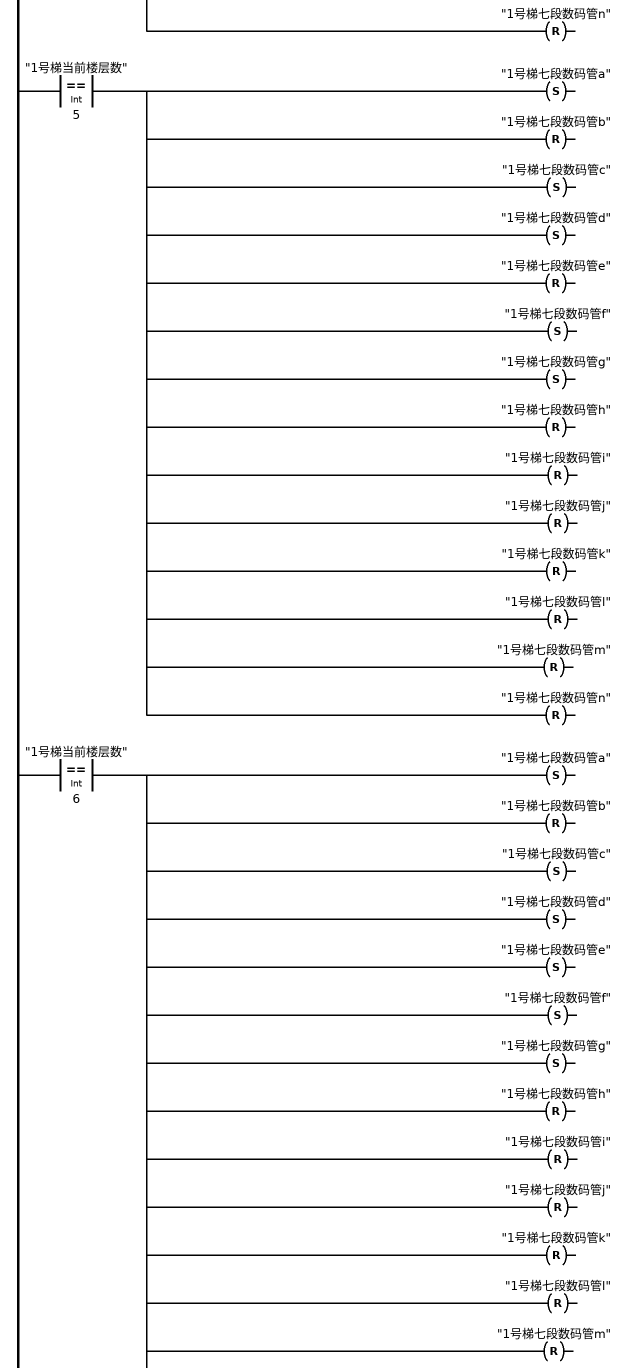
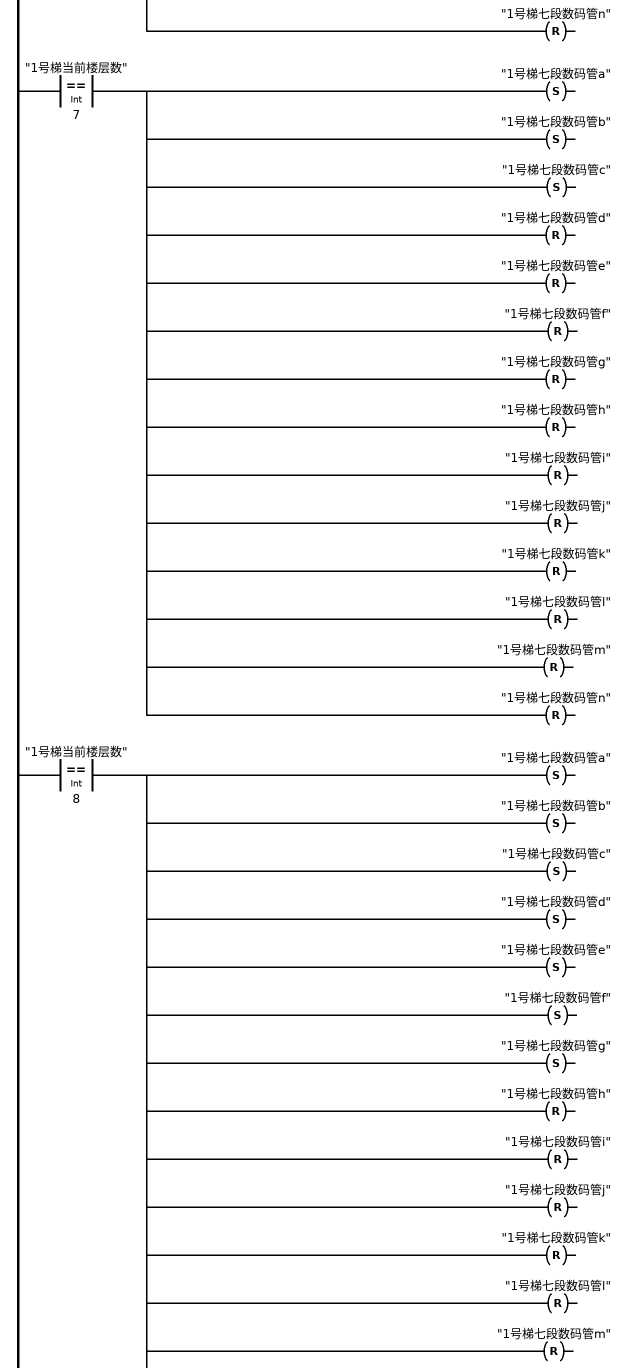
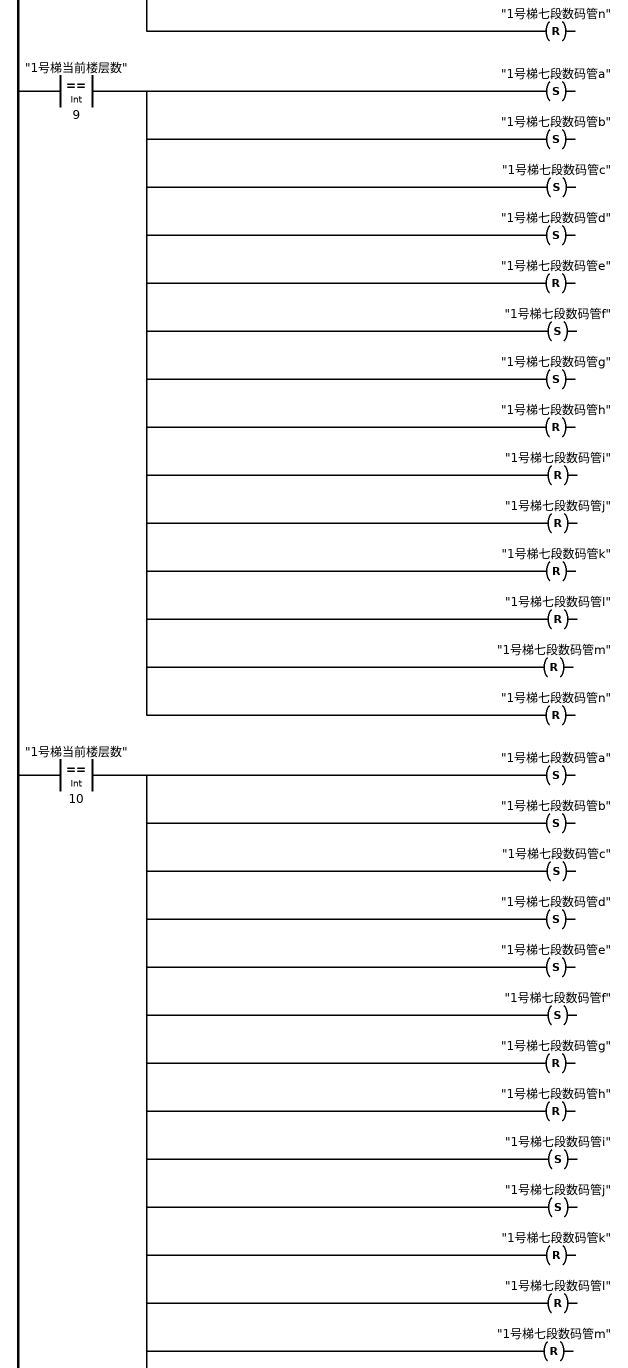
